LIN {X 0,Y 680.523,Z 319.435,A -85,B 0,C 180,E1 25560.421,E2 25560.421} C_VEL
LIN {X 0,Y 680.503,Z 319.465,A -85,B 0,C 180,E1 25557.305,E2 25557.305} C_VEL
LIN {X 0,Y 680.521,Z 319.439,A -85,B 0,C 180,E1 25554.266,E2 25554.266} C_VEL
LIN {X 0,Y 680.497,Z 319.465,A -85,B 0,C 180,E1 25551.21,E2 25551.21} C_VEL
LIN {X 0,Y 680.519,Z 319.439,A -85,B 0,C 180,E1 25548.215,E2 25548.215} C_VEL
LIN {X 0,Y 680.491,Z 319.465,A -85,B 0,C 180,E1 25545.1,E2 25545.1} C_VEL
LIN {X 0,Y 680.502,Z 319.438,A -85,B 0,C 180,E1 25542.198,E2 25542.198} C_VEL
LIN {X 0,Y 680.491,Z 319.464,A -85,B 0,C 180,E1 25539.08,E2 25539.08} C_VEL
LIN {X 0,Y 680.47,Z 319.444,A -85,B 0,C 180,E1 25536.35,E2 25536.35} C_VEL
LIN {X 0,Y 680.519,Z 319.455,A -85,B 0,C 180,E1 25533.281,E2 25533.281} C_VEL
LIN {X 0,Y 680.458,Z 319.465,A -85,B 0,C 180,E1 25530.51,E2 25530.51} C_VEL
LIN {X 0,Y 680.498,Z 319.446,A -85,B 0,C 180,E1 25527.766,E2 25527.766} C_VEL
LIN {X 0,Y 680.46,Z 319.462,A -85,B 0,C 180,E1 25524.726,E2 25524.726} C_VEL
LIN {X 0,Y 680.444,Z 319.466,A -85,B 0,C 180,E1 25522.21,E2 25522.21} C_VEL
LIN {X 0,Y 680.534,Z 319.527,A -85,B 0,C 180,E1 25519.314,E2 25519.314} C_VEL
LIN {X 0,Y 680.713,Z 320.476,A -85,B 0,C 180,E1 25519.153,E2 25519.153} C_VEL
LIN {X 0,Y 688.87,Z 336.842,A -85,B 0,C 180,E1 25517.211,E2 25517.211} C_VEL
LIN {X 0,Y 695.472,Z 350.637,A -85,B 0,C 180,E1 25515.703,E2 25515.703} C_VEL
LIN {X 0,Y 696.705,Z 353.093,A -85,B 0,C 180,E1 25515.558,E2 25515.558} C_VEL
LIN {X 0,Y 700.836,Z 371.518,A -85,B 0,C 180,E1 25514.953,E2 25514.953} C_VEL
LIN {X 0,Y 698.449,Z 583.894,A -85,B 0,C 180,E1 25512.191,E2 25512.191} C_VEL
LIN {X 0,Y 696.12,Z 808.395,A -85,B 0,C 180,E1 25509.364,E2 25509.364} C_VEL
LIN {X 0,Y 695.539,Z 840.013,A -85,B 0,C 180,E1 25508.911,E2 25508.911} C_VEL
LIN {X 0,Y 694.786,Z 865.208,A -85,B 0,C 180,E1 25508.397,E2 25508.397} C_VEL
LIN {X 0,Y 693.902,Z 890.782,A -85,B 0,C 180,E1 25507.726,E2 25507.726} C_VEL
LIN {X 0,Y 692.784,Z 917.463,A -85,B 0,C 180,E1 25506.847,E2 25506.847} C_VEL
LIN {X 0,Y 691.789,Z 938.354,A -85,B 0,C 180,E1 25506.033,E2 25506.033} C_VEL
LIN {X 0,Y 690.754,Z 958.67,A -85,B 0,C 180,E1 25505.129,E2 25505.129} C_VEL
LIN {X 0,Y 689.673,Z 978.671,A -85,B 0,C 180,E1 25504.122,E2 25504.122} C_VEL
LIN {X 0,Y 688.521,Z 999.46,A -85,B 0,C 180,E1 25502.946,E2 25502.946} C_VEL
LIN {X 0,Y 687.068,Z 1024.247,A -85,B 0,C 180,E1 25501.35,E2 25501.35} C_VEL
LIN {X 0,Y 685.992,Z 1043.448,A -85,B 0,C 180,E1 25499.948,E2 25499.948} C_VEL
LIN {X 0,Y 684.974,Z 1061.822,A -85,B 0,C 180,E1 25498.464,E2 25498.464} C_VEL
LIN {X 0,Y 683.767,Z 1083.482,A -85,B 0,C 180,E1 25496.498,E2 25496.498} C_VEL
LIN {X 0,Y 682.983,Z 1099.693,A -85,B 0,C 180,E1 25494.845,E2 25494.845} C_VEL
LIN {X 0,Y 682.191,Z 1116.49,A -85,B 0,C 180,E1 25492.946,E2 25492.946} C_VEL
LIN {X 0,Y 681.497,Z 1132.896,A -85,B 0,C 180,E1 25490.835,E2 25490.835} C_VEL
LIN {X 0,Y 681.036,Z 1145.574,A -85,B 0,C 180,E1 25489,E2 25489} C_VEL
LIN {X 0,Y 680.644,Z 1157.898,A -85,B 0,C 180,E1 25486.992,E2 25486.992} C_VEL
LIN {X 0,Y 680.336,Z 1169.839,A -85,B 0,C 180,E1 25484.729,E2 25484.729} C_VEL
LIN {X 0,Y 680.158,Z 1178.438,A -85,B 0,C 180,E1 25482.825,E2 25482.825} C_VEL
LIN {X 0,Y 680.019,Z 1186.223,A -85,B 0,C 180,E1 25480.82,E2 25480.82} C_VEL
LIN {X 0,Y 679.964,Z 1193.354,A -85,B 0,C 180,E1 25478.541,E2 25478.541} C_VEL
LIN {X 0,Y 679.926,Z 1198.83,A -85,B 0,C 180,E1 25476.216,E2 25476.216} C_VEL
LIN {X 0,Y 679.913,Z 1202.374,A -85,B 0,C 180,E1 25474.048,E2 25474.048} C_VEL
LIN {X 0,Y 679.907,Z 1204.494,A -85,B 0,C 180,E1 25471.77,E2 25471.77} C_VEL
LIN {X 0,Y 679.891,Z 1204.872,A -85,B 0,C 180,E1 25469.494,E2 25469.494} C_VEL
LIN {X 0,Y 679.907,Z 1203.956,A -85,B 0,C 180,E1 25467.471,E2 25467.471} C_VEL
LIN {X 0,Y 679.911,Z 1201.427,A -85,B 0,C 180,E1 25465.276,E2 25465.276} C_VEL
LIN {X 0,Y 679.933,Z 1197.151,A -85,B 0,C 180,E1 25462.989,E2 25462.989} C_VEL
LIN {X 0,Y 679.979,Z 1191.384,A -85,B 0,C 180,E1 25460.777,E2 25460.777} C_VEL
LIN {X 0,Y 680.067,Z 1184.276,A -85,B 0,C 180,E1 25458.637,E2 25458.637} C_VEL
LIN {X 0,Y 680.241,Z 1173.935,A -85,B 0,C 180,E1 25456.137,E2 25456.137} C_VEL
LIN {X 0,Y 680.464,Z 1164.535,A -85,B 0,C 180,E1 25454.226,E2 25454.226} C_VEL
LIN {X 0,Y 680.75,Z 1154.226,A -85,B 0,C 180,E1 25452.388,E2 25452.388} C_VEL
LIN {X 0,Y 681.151,Z 1141.935,A -85,B 0,C 180,E1 25450.446,E2 25450.446} C_VEL
LIN {X 0,Y 681.795,Z 1125.468,A -85,B 0,C 180,E1 25448.177,E2 25448.177} C_VEL
LIN {X 0,Y 682.44,Z 1111.066,A -85,B 0,C 180,E1 25446.423,E2 25446.423} C_VEL
LIN {X 0,Y 683.272,Z 1093.714,A -85,B 0,C 180,E1 25444.518,E2 25444.518} C_VEL
LIN {X 0,Y 684.267,Z 1074.727,A -85,B 0,C 180,E1 25442.679,E2 25442.679} C_VEL
LIN {X 0,Y 685.157,Z 1057.943,A -85,B 0,C 180,E1 25441.211,E2 25441.211} C_VEL
LIN {X 0,Y 686.262,Z 1038.582,A -85,B 0,C 180,E1 25439.679,E2 25439.679} C_VEL
LIN {X 0,Y 687.621,Z 1015.166,A -85,B 0,C 180,E1 25438.042,E2 25438.042} C_VEL
LIN {X 0,Y 688.735,Z 995.434,A -85,B 0,C 180,E1 25436.817,E2 25436.817} C_VEL
LIN {X 0,Y 689.842,Z 975.499,A -85,B 0,C 180,E1 25435.709,E2 25435.709} C_VEL
LIN {X 0,Y 691.119,Z 951.675,A -85,B 0,C 180,E1 25434.539,E2 25434.539} C_VEL
LIN {X 0,Y 692.336,Z 926.405,A -85,B 0,C 180,E1 25433.486,E2 25433.486} C_VEL
LIN {X 0,Y 693.318,Z 904.116,A -85,B 0,C 180,E1 25432.694,E2 25432.694} C_VEL
LIN {X 0,Y 694.253,Z 881.033,A -85,B 0,C 180,E1 25432.001,E2 25432.001} C_VEL
LIN {X 0,Y 695.166,Z 854.064,A -85,B 0,C 180,E1 25431.355,E2 25431.355} C_VEL
LIN {X 0,Y 695.823,Z 827.013,A -85,B 0,C 180,E1 25430.882,E2 25430.882} C_VEL
LIN {X 0,Y 698.199,Z 606.762,A -85,B 0,C 180,E1 25428.101,E2 25428.101} C_VEL
LIN {X 0,Y 700.451,Z 403.611,A -85,B 0,C 180,E1 25425.47,E2 25425.47} C_VEL
LIN {X 0,Y 700.679,Z 370.058,A -85,B 0,C 180,E1 25425.014,E2 25425.014} C_VEL
LIN {X 0,Y 696.204,Z 351.824,A -85,B 0,C 180,E1 25424.382,E2 25424.382} C_VEL
LIN {X 0,Y 694.705,Z 349.075,A -85,B 0,C 180,E1 25424.157,E2 25424.157} C_VEL
LIN {X 0,Y 686.31,Z 331.797,A -85,B 0,C 180,E1 25422.194,E2 25422.194} C_VEL
LIN {X 0,Y 681.971,Z 323.226,A -85,B 0,C 180,E1 25421.172,E2 25421.172} C_VEL
LIN {X 0,Y 680.561,Z 319.709,A -85,B 0,C 180,E1 25420.745,E2 25420.745} C_VEL
LIN {X 0,Y 680.447,Z 319.469,A -85,B 0,C 180,E1 25417.897,E2 25417.897} C_VEL
LIN {X 0,Y 680.453,Z 319.462,A -85,B 0,C 180,E1 25415.36,E2 25415.36} C_VEL
LIN {X 0,Y 680.511,Z 319.443,A -85,B 0,C 180,E1 25412.333,E2 25412.333} C_VEL
LIN {X 0,Y 680.457,Z 319.465,A -85,B 0,C 180,E1 25409.553,E2 25409.553} C_VEL
LIN {X 0,Y 680.502,Z 319.454,A -85,B 0,C 180,E1 25406.814,E2 25406.814} C_VEL
LIN {X 0,Y 680.474,Z 319.444,A -85,B 0,C 180,E1 25403.733,E2 25403.733} C_VEL
LIN {X 0,Y 680.48,Z 319.464,A -85,B 0,C 180,E1 25401.01,E2 25401.01} C_VEL
LIN {X 0,Y 680.509,Z 319.438,A -85,B 0,C 180,E1 25397.884,E2 25397.884} C_VEL
LIN {X 0,Y 680.481,Z 319.465,A -85,B 0,C 180,E1 25394.988,E2 25394.988} C_VEL
LIN {X 0,Y 680.522,Z 319.437,A -85,B 0,C 180,E1 25391.957,E2 25391.957} C_VEL
LIN {X 0,Y 680.483,Z 319.463,A -85,B 0,C 180,E1 25389.046,E2 25389.046} C_VEL
LIN {X 0,Y 680.517,Z 319.437,A -85,B 0,C 180,E1 25386.157,E2 25386.157} C_VEL
LIN {X 0,Y 680.493,Z 319.46,A -85,B 0,C 180,E1 25383.117,E2 25383.117} C_VEL
LIN {X 0,Y 680.518,Z 319.436,A -85,B 0,C 180,E1 25380.168,E2 25380.168} C_VEL
LIN {X 0,Y 680.504,Z 319.457,A -85,B 0,C 180,E1 25377.116,E2 25377.116} C_VEL
LIN {X 0,Y 680.515,Z 319.436,A -85,B 0,C 180,E1 25374.097,E2 25374.097} C_VEL
LIN {X 0,Y 680.513,Z 319.455,A -85,B 0,C 180,E1 25371.04,E2 25371.04} C_VEL
LIN {X 0,Y 680.514,Z 319.438,A -85,B 0,C 180,E1 25368.043,E2 25368.043} C_VEL
LIN {X 0,Y 680.523,Z 319.455,A -85,B 0,C 180,E1 25365.013,E2 25365.013} C_VEL
LIN {X 0,Y 680.509,Z 319.44,A -85,B 0,C 180,E1 25361.924,E2 25361.924} C_VEL
LIN {X 0,Y 680.526,Z 319.457,A -85,B 0,C 180,E1 25358.901,E2 25358.901} C_VEL
LIN {X 0,Y 680.503,Z 319.444,A -85,B 0,C 180,E1 25355.798,E2 25355.798} C_VEL
LIN {X 0,Y 680.523,Z 319.457,A -85,B 0,C 180,E1 25352.737,E2 25352.737} C_VEL
LIN {X 0,Y 680.495,Z 319.462,A -85,B 0,C 180,E1 25349.638,E2 25349.638} C_VEL
LIN {X 0,Y 680.486,Z 319.466,A -85,B 0,C 180,E1 25349.46,E2 25349.46} C_VEL
LIN {X 0,Y 679.484,Z 319.589,A -85,B 0,C 180,E1 25348.811,E2 25348.811} C_VEL
LIN {X 0,Y 673.087,Z 320.364,A -85,B 0,C 180,E1 25346.994,E2 25346.994} C_VEL
LIN {X 0,Y 672.583,Z 320.425,A -85,B 0,C 180,E1 25346.521,E2 25346.521} C_VEL
LIN {X 0,Y 672.547,Z 320.44,A -85,B 0,C 180,E1 25343.509,E2 25343.509} C_VEL
LIN {X 0,Y 672.564,Z 320.456,A -85,B 0,C 180,E1 25340.594,E2 25340.594} C_VEL
LIN {X 0,Y 672.618,Z 320.685,A -85,B 0,C 180,E1 25338.341,E2 25338.341} C_VEL
LIN {X 0,Y 674.146,Z 324.296,A -85,B 0,C 180,E1 25337.867,E2 25337.867} C_VEL
LIN {X 0,Y 680.947,Z 338.516,A -85,B 0,C 180,E1 25336.126,E2 25336.126} C_VEL
LIN {X 0,Y 687.645,Z 353.245,A -85,B 0,C 180,E1 25334.442,E2 25334.442} C_VEL
LIN {X 0,Y 688.188,Z 354.8,A -85,B 0,C 180,E1 25334.283,E2 25334.283} C_VEL
LIN {X 0,Y 686.298,Z 396.404,A -85,B 0,C 180,E1 25331.484,E2 25331.484} C_VEL
LIN {X 0,Y 690.87,Z 417.786,A -85,B 0,C 180,E1 25330.837,E2 25330.837} C_VEL
LIN {X 0,Y 688.26,Z 661.816,A -85,B 0,C 180,E1 25327.794,E2 25327.794} C_VEL
LIN {X 0,Y 686.473,Z 830.346,A -85,B 0,C 180,E1 25325.723,E2 25325.723} C_VEL
LIN {X 0,Y 685.847,Z 856.635,A -85,B 0,C 180,E1 25325.262,E2 25325.262} C_VEL
LIN {X 0,Y 685.019,Z 880.355,A -85,B 0,C 180,E1 25324.692,E2 25324.692} C_VEL
LIN {X 0,Y 684.217,Z 900.856,A -85,B 0,C 180,E1 25324.085,E2 25324.085} C_VEL
LIN {X 0,Y 683.164,Z 924.808,A -85,B 0,C 180,E1 25323.238,E2 25323.238} C_VEL
LIN {X 0,Y 681.985,Z 948.429,A -85,B 0,C 180,E1 25322.224,E2 25322.224} C_VEL
LIN {X 0,Y 680.95,Z 968.049,A -85,B 0,C 180,E1 25321.255,E2 25321.255} C_VEL
LIN {X 0,Y 679.738,Z 990.237,A -85,B 0,C 180,E1 25320.009,E2 25320.009} C_VEL
LIN {X 0,Y 678.458,Z 1011.622,A -85,B 0,C 180,E1 25318.618,E2 25318.618} C_VEL
LIN {X 0,Y 677.441,Z 1029.893,A -85,B 0,C 180,E1 25317.282,E2 25317.282} C_VEL
LIN {X 0,Y 676.241,Z 1051.038,A -85,B 0,C 180,E1 25315.532,E2 25315.532} C_VEL
LIN {X 0,Y 675.373,Z 1067.296,A -85,B 0,C 180,E1 25314.01,E2 25314.01} C_VEL
LIN {X 0,Y 674.523,Z 1084.551,A -85,B 0,C 180,E1 25312.21,E2 25312.21} C_VEL
LIN {X 0,Y 673.77,Z 1100.533,A -85,B 0,C 180,E1 25310.297,E2 25310.297} C_VEL
LIN {X 0,Y 673.204,Z 1114.293,A -85,B 0,C 180,E1 25308.443,E2 25308.443} C_VEL
LIN {X 0,Y 672.711,Z 1127.982,A -85,B 0,C 180,E1 25306.315,E2 25306.315} C_VEL
LIN {X 0,Y 672.442,Z 1137.959,A -85,B 0,C 180,E1 25304.531,E2 25304.531} C_VEL
LIN {X 0,Y 672.2,Z 1148.015,A -85,B 0,C 180,E1 25302.456,E2 25302.456} C_VEL
LIN {X 0,Y 672.044,Z 1156.61,A -85,B 0,C 180,E1 25300.285,E2 25300.285} C_VEL
LIN {X 0,Y 671.973,Z 1162.516,A -85,B 0,C 180,E1 25298.471,E2 25298.471} C_VEL
LIN {X 0,Y 671.925,Z 1167.459,A -85,B 0,C 180,E1 25296.58,E2 25296.58} C_VEL
LIN {X 0,Y 671.909,Z 1171.777,A -85,B 0,C 180,E1 25294.267,E2 25294.267} C_VEL
LIN {X 0,Y 671.913,Z 1173.902,A -85,B 0,C 180,E1 25292.388,E2 25292.388} C_VEL
LIN {X 0,Y 671.892,Z 1174.837,A -85,B 0,C 180,E1 25290.597,E2 25290.597} C_VEL
LIN {X 0,Y 671.91,Z 1174.637,A -85,B 0,C 180,E1 25288.551,E2 25288.551} C_VEL
LIN {X 0,Y 671.897,Z 1172.688,A -85,B 0,C 180,E1 25286.331,E2 25286.331} C_VEL
LIN {X 0,Y 671.909,Z 1169.91,A -85,B 0,C 180,E1 25284.535,E2 25284.535} C_VEL
LIN {X 0,Y 671.944,Z 1166.023,A -85,B 0,C 180,E1 25282.734,E2 25282.734} C_VEL
LIN {X 0,Y 672.007,Z 1159.937,A -85,B 0,C 180,E1 25280.573,E2 25280.573} C_VEL
LIN {X 0,Y 672.123,Z 1151.993,A -85,B 0,C 180,E1 25278.415,E2 25278.415} C_VEL
LIN {X 0,Y 672.271,Z 1144.372,A -85,B 0,C 180,E1 25276.672,E2 25276.672} C_VEL
LIN {X 0,Y 672.556,Z 1133.669,A -85,B 0,C 180,E1 25274.567,E2 25274.567} C_VEL
LIN {X 0,Y 672.937,Z 1121.399,A -85,B 0,C 180,E1 25272.534,E2 25272.534} C_VEL
LIN {X 0,Y 673.404,Z 1109.186,A -85,B 0,C 180,E1 25270.754,E2 25270.754} C_VEL
LIN {X 0,Y 674.119,Z 1092.876,A -85,B 0,C 180,E1 25268.668,E2 25268.668} C_VEL
LIN {X 0,Y 674.819,Z 1077.786,A -85,B 0,C 180,E1 25266.973,E2 25266.973} C_VEL
LIN {X 0,Y 675.804,Z 1059.628,A -85,B 0,C 180,E1 25265.154,E2 25265.154} C_VEL
LIN {X 0,Y 676.807,Z 1040.8,A -85,B 0,C 180,E1 25263.503,E2 25263.503} C_VEL
LIN {X 0,Y 677.936,Z 1021.383,A -85,B 0,C 180,E1 25261.982,E2 25261.982} C_VEL
LIN {X 0,Y 679.191,Z 999.206,A -85,B 0,C 180,E1 25260.466,E2 25260.466} C_VEL
LIN {X 0,Y 680.323,Z 978.831,A -85,B 0,C 180,E1 25259.239,E2 25259.239} C_VEL
LIN {X 0,Y 681.679,Z 954.593,A -85,B 0,C 180,E1 25257.975,E2 25257.975} C_VEL
LIN {X 0,Y 682.736,Z 933.698,A -85,B 0,C 180,E1 25257.039,E2 25257.039} C_VEL
LIN {X 0,Y 683.65,Z 914.34,A -85,B 0,C 180,E1 25256.287,E2 25256.287} C_VEL
LIN {X 0,Y 684.698,Z 889.896,A -85,B 0,C 180,E1 25255.48,E2 25255.48} C_VEL
LIN {X 0,Y 685.52,Z 864.903,A -85,B 0,C 180,E1 25254.831,E2 25254.831} C_VEL
LIN {X 0,Y 686.17,Z 842.781,A -85,B 0,C 180,E1 25254.384,E2 25254.384} C_VEL
LIN {X 0,Y 686.74,Z 813.095,A -85,B 0,C 180,E1 25253.957,E2 25253.957} C_VEL
LIN {X 0,Y 689.172,Z 573.619,A -85,B 0,C 180,E1 25251.027,E2 25251.027} C_VEL
LIN {X 0,Y 690.784,Z 416.524,A -85,B 0,C 180,E1 25249.05,E2 25249.05} C_VEL
LIN {X 0,Y 686.265,Z 396.184,A -85,B 0,C 180,E1 25248.417,E2 25248.417} C_VEL
LIN {X 0,Y 688.188,Z 354.854,A -85,B 0,C 180,E1 25245.631,E2 25245.631} C_VEL
LIN {X 0,Y 683.619,Z 344.296,A -85,B 0,C 180,E1 25244.459,E2 25244.459} C_VEL
LIN {X 0,Y 678.067,Z 332.508,A -85,B 0,C 180,E1 25243.059,E2 25243.059} C_VEL
LIN {X 0,Y 673.851,Z 323.857,A -85,B 0,C 180,E1 25241.979,E2 25241.979} C_VEL
LIN {X 0,Y 672.598,Z 320.636,A -85,B 0,C 180,E1 25241.546,E2 25241.546} C_VEL
LIN {X 0,Y 672.527,Z 320.454,A -85,B 0,C 180,E1 25238.751,E2 25238.751} C_VEL
LIN {X 0,Y 672.587,Z 320.447,A -85,B 0,C 180,E1 25235.855,E2 25235.855} C_VEL
LIN {X 0,Y 672.537,Z 320.433,A -85,B 0,C 180,E1 25232.86,E2 25232.86} C_VEL
LIN {X 0,Y 672.586,Z 320.436,A -85,B 0,C 180,E1 25229.968,E2 25229.968} C_VEL
LIN {X 0,Y 672.554,Z 320.449,A -85,B 0,C 180,E1 25226.87,E2 25226.87} C_VEL
LIN {X 0,Y 672.579,Z 320.427,A -85,B 0,C 180,E1 25223.897,E2 25223.897} C_VEL
LIN {X 0,Y 672.562,Z 320.449,A -85,B 0,C 180,E1 25220.754,E2 25220.754} C_VEL
LIN {X 0,Y 672.58,Z 320.428,A -85,B 0,C 180,E1 25217.744,E2 25217.744} C_VEL
LIN {X 0,Y 672.567,Z 320.447,A -85,B 0,C 180,E1 25214.64,E2 25214.64} C_VEL
LIN {X 0,Y 672.575,Z 320.431,A -85,B 0,C 180,E1 25211.567,E2 25211.567} C_VEL
LIN {X 0,Y 672.572,Z 320.445,A -85,B 0,C 180,E1 25208.464,E2 25208.464} C_VEL
LIN {X 0,Y 672.57,Z 320.431,A -85,B 0,C 180,E1 25205.46,E2 25205.46} C_VEL
LIN {X 0,Y 672.579,Z 320.445,A -85,B 0,C 180,E1 25202.386,E2 25202.386} C_VEL
LIN {X 0,Y 672.564,Z 320.432,A -85,B 0,C 180,E1 25199.319,E2 25199.319} C_VEL
LIN {X 0,Y 672.582,Z 320.447,A -85,B 0,C 180,E1 25196.249,E2 25196.249} C_VEL
LIN {X 0,Y 672.553,Z 320.433,A -85,B 0,C 180,E1 25193.169,E2 25193.169} C_VEL
LIN {X 0,Y 672.585,Z 320.446,A -85,B 0,C 180,E1 25190.156,E2 25190.156} C_VEL
LIN {X 0,Y 672.551,Z 320.434,A -85,B 0,C 180,E1 25187.114,E2 25187.114} C_VEL
LIN {X 0,Y 672.57,Z 320.448,A -85,B 0,C 180,E1 25184.213,E2 25184.213} C_VEL
LIN {X 0,Y 672.549,Z 320.438,A -85,B 0,C 180,E1 25181.089,E2 25181.089} C_VEL
LIN {X 0,Y 672.545,Z 320.448,A -85,B 0,C 180,E1 25178.272,E2 25178.272} C_VEL
LIN {X 0,Y 672.552,Z 320.451,A -85,B 0,C 180,E1 25175.077,E2 25175.077} C_VEL
LIN {X 0,Y 672.523,Z 320.437,A -85,B 0,C 180,E1 25172.362,E2 25172.362} C_VEL
LIN {X 0,Y 672.59,Z 320.454,A -85,B 0,C 180,E1 25169.4,E2 25169.4} C_VEL
LIN {X 0,Y 672.513,Z 320.445,A -85,B 0,C 180,E1 25166.52,E2 25166.52} C_VEL
LIN {X 0,Y 672.535,Z 320.433,A -85,B 0,C 180,E1 25163.826,E2 25163.826} C_VEL
LIN {X 0,Y 672.516,Z 320.44,A -85,B 0,C 180,E1 25160.7,E2 25160.7} C_VEL
LIN {X 0,Y 672.546,Z 320.693,A -85,B 0,C 180,E1 25159.954,E2 25159.954} C_VEL
LIN {X 0,Y 674.168,Z 324.332,A -85,B 0,C 180,E1 25159.487,E2 25159.487} C_VEL
LIN {X 0,Y 683.149,Z 342.282,A -85,B 0,C 180,E1 25157.338,E2 25157.338} C_VEL
LIN {X 0,Y 687.378,Z 350.803,A -85,B 0,C 180,E1 25156.395,E2 25156.395} C_VEL
LIN {X 0,Y 691.603,Z 357.548,A -85,B 0,C 180,E1 25155.925,E2 25155.925} C_VEL
LIN {X 0,Y 695.139,Z 373.566,A -85,B 0,C 180,E1 25155.394,E2 25155.394} C_VEL
LIN {X 0,Y 692.485,Z 586.297,A -85,B 0,C 180,E1 25152.607,E2 25152.607} C_VEL
LIN {X 0,Y 689.906,Z 810.507,A -85,B 0,C 180,E1 25149.761,E2 25149.761} C_VEL
LIN {X 0,Y 689.269,Z 840.637,A -85,B 0,C 180,E1 25149.32,E2 25149.32} C_VEL
LIN {X 0,Y 688.472,Z 865.187,A -85,B 0,C 180,E1 25148.815,E2 25148.815} C_VEL
LIN {X 0,Y 687.488,Z 890.734,A -85,B 0,C 180,E1 25148.142,E2 25148.142} C_VEL
LIN {X 0,Y 686.225,Z 918.038,A -85,B 0,C 180,E1 25147.235,E2 25147.235} C_VEL
LIN {X 0,Y 685.095,Z 939.48,A -85,B 0,C 180,E1 25146.39,E2 25146.39} C_VEL
LIN {X 0,Y 683.956,Z 959.717,A -85,B 0,C 180,E1 25145.477,E2 25145.477} C_VEL
LIN {X 0,Y 682.726,Z 980.329,A -85,B 0,C 180,E1 25144.424,E2 25144.424} C_VEL
LIN {X 0,Y 681.2,Z 1004.932,A -85,B 0,C 180,E1 25142.994,E2 25142.994} C_VEL
LIN {X 0,Y 679.764,Z 1026.915,A -85,B 0,C 180,E1 25141.527,E2 25141.527} C_VEL
LIN {X 0,Y 678.597,Z 1045.715,A -85,B 0,C 180,E1 25140.125,E2 25140.125} C_VEL
LIN {X 0,Y 677.318,Z 1066.77,A -85,B 0,C 180,E1 25138.376,E2 25138.376} C_VEL
LIN {X 0,Y 676.138,Z 1085.454,A -85,B 0,C 180,E1 25136.62,E2 25136.62} C_VEL
LIN {X 0,Y 675.284,Z 1101.391,A -85,B 0,C 180,E1 25134.96,E2 25134.96} C_VEL
LIN {X 0,Y 674.295,Z 1120.136,A -85,B 0,C 180,E1 25132.769,E2 25132.769} C_VEL
LIN {X 0,Y 673.636,Z 1134.462,A -85,B 0,C 180,E1 25130.869,E2 25130.869} C_VEL
LIN {X 0,Y 673.123,Z 1147.168,A -85,B 0,C 180,E1 25128.984,E2 25128.984} C_VEL
LIN {X 0,Y 672.64,Z 1160.813,A -85,B 0,C 180,E1 25126.672,E2 25126.672} C_VEL
LIN {X 0,Y 672.362,Z 1171.072,A -85,B 0,C 180,E1 25124.644,E2 25124.644} C_VEL
LIN {X 0,Y 672.176,Z 1179.154,A -85,B 0,C 180,E1 25122.805,E2 25122.805} C_VEL
LIN {X 0,Y 672.03,Z 1186.719,A -85,B 0,C 180,E1 25120.805,E2 25120.805} C_VEL
LIN {X 0,Y 671.969,Z 1193.595,A -85,B 0,C 180,E1 25118.557,E2 25118.557} C_VEL
LIN {X 0,Y 671.928,Z 1198.937,A -85,B 0,C 180,E1 25116.236,E2 25116.236} C_VEL
LIN {X 0,Y 671.915,Z 1202.371,A -85,B 0,C 180,E1 25114.096,E2 25114.096} C_VEL
LIN {X 0,Y 671.907,Z 1204.494,A -85,B 0,C 180,E1 25111.791,E2 25111.791} C_VEL
LIN {X 0,Y 671.891,Z 1204.872,A -85,B 0,C 180,E1 25109.488,E2 25109.488} C_VEL
LIN {X 0,Y 671.907,Z 1203.953,A -85,B 0,C 180,E1 25107.441,E2 25107.441} C_VEL
LIN {X 0,Y 671.914,Z 1201.427,A -85,B 0,C 180,E1 25105.22,E2 25105.22} C_VEL
LIN {X 0,Y 671.941,Z 1197.151,A -85,B 0,C 180,E1 25102.905,E2 25102.905} C_VEL
LIN {X 0,Y 671.991,Z 1191.381,A -85,B 0,C 180,E1 25100.666,E2 25100.666} C_VEL
LIN {X 0,Y 672.09,Z 1184.276,A -85,B 0,C 180,E1 25098.501,E2 25098.501} C_VEL
LIN {X 0,Y 672.277,Z 1174.339,A -85,B 0,C 180,E1 25096.058,E2 25096.058} C_VEL
LIN {X 0,Y 672.534,Z 1164.537,A -85,B 0,C 180,E1 25094.035,E2 25094.035} C_VEL
LIN {X 0,Y 672.865,Z 1154.228,A -85,B 0,C 180,E1 25092.175,E2 25092.175} C_VEL
LIN {X 0,Y 673.32,Z 1141.937,A -85,B 0,C 180,E1 25090.21,E2 25090.21} C_VEL
LIN {X 0,Y 674.025,Z 1125.804,A -85,B 0,C 180,E1 25087.956,E2 25087.956} C_VEL
LIN {X 0,Y 674.751,Z 1111.068,A -85,B 0,C 180,E1 25086.137,E2 25086.137} C_VEL
LIN {X 0,Y 675.713,Z 1093.715,A -85,B 0,C 180,E1 25084.212,E2 25084.212} C_VEL
LIN {X 0,Y 676.819,Z 1074.319,A -85,B 0,C 180,E1 25082.314,E2 25082.314} C_VEL
LIN {X 0,Y 677.817,Z 1057.656,A -85,B 0,C 180,E1 25080.845,E2 25080.845} C_VEL
LIN {X 0,Y 679.091,Z 1037.972,A -85,B 0,C 180,E1 25079.275,E2 25079.275} C_VEL
LIN {X 0,Y 680.589,Z 1014.441,A -85,B 0,C 180,E1 25077.622,E2 25077.622} C_VEL
LIN {X 0,Y 681.824,Z 994.634,A -85,B 0,C 180,E1 25076.386,E2 25076.386} C_VEL
LIN {X 0,Y 683.132,Z 973.152,A -85,B 0,C 180,E1 25075.192,E2 25075.192} C_VEL
LIN {X 0,Y 684.732,Z 946.206,A -85,B 0,C 180,E1 25073.899,E2 25073.899} C_VEL
LIN {X 0,Y 685.854,Z 925.016,A -85,B 0,C 180,E1 25073.027,E2 25073.027} C_VEL
LIN {X 0,Y 686.854,Z 904.042,A -85,B 0,C 180,E1 25072.279,E2 25072.279} C_VEL
LIN {X 0,Y 687.876,Z 880.995,A -85,B 0,C 180,E1 25071.584,E2 25071.584} C_VEL
LIN {X 0,Y 688.887,Z 854.024,A -85,B 0,C 180,E1 25070.935,E2 25070.935} C_VEL
LIN {X 0,Y 689.603,Z 827.087,A -85,B 0,C 180,E1 25070.462,E2 25070.462} C_VEL
LIN {X 0,Y 692.206,Z 609.542,A -85,B 0,C 180,E1 25067.692,E2 25067.692} C_VEL
LIN {X 0,Y 694.706,Z 406.307,A -85,B 0,C 180,E1 25065.04,E2 25065.04} C_VEL
LIN {X 0,Y 694.99,Z 372.179,A -85,B 0,C 180,E1 25064.574,E2 25064.574} C_VEL
LIN {X 0,Y 691.173,Z 356.512,A -85,B 0,C 180,E1 25064.023,E2 25064.023} C_VEL
LIN {X 0,Y 686.793,Z 349.864,A -85,B 0,C 180,E1 25063.522,E2 25063.522} C_VEL
LIN {X 0,Y 678.81,Z 333.538,A -85,B 0,C 180,E1 25061.631,E2 25061.631} C_VEL
LIN {X 0,Y 674.765,Z 325.222,A -85,B 0,C 180,E1 25060.637,E2 25060.637} C_VEL
LIN {X 0,Y 672.758,Z 321.621,A -85,B 0,C 180,E1 25060.169,E2 25060.169} C_VEL
LIN {X 0,Y 672.522,Z 320.554,A -85,B 0,C 180,E1 25059.999,E2 25059.999} C_VEL
LIN {X 0,Y 672.508,Z 320.443,A -85,B 0,C 180,E1 25057.444,E2 25057.444} C_VEL
LIN {X 0,Y 672.573,Z 320.452,A -85,B 0,C 180,E1 25054.402,E2 25054.402} C_VEL
LIN {X 0,Y 672.513,Z 320.448,A -85,B 0,C 180,E1 25051.558,E2 25051.558} C_VEL
LIN {X 0,Y 672.566,Z 320.432,A -85,B 0,C 180,E1 25048.796,E2 25048.796} C_VEL
LIN {X 0,Y 672.533,Z 320.454,A -85,B 0,C 180,E1 25045.715,E2 25045.715} C_VEL
LIN {X 0,Y 672.545,Z 320.429,A -85,B 0,C 180,E1 25042.925,E2 25042.925} C_VEL
LIN {X 0,Y 672.55,Z 320.447,A -85,B 0,C 180,E1 25039.724,E2 25039.724} C_VEL
LIN {X 0,Y 672.549,Z 320.434,A -85,B 0,C 180,E1 25036.853,E2 25036.853} C_VEL
LIN {X 0,Y 672.564,Z 320.44,A -85,B 0,C 180,E1 25033.673,E2 25033.673} C_VEL
LIN {X 0,Y 672.562,Z 320.438,A -85,B 0,C 180,E1 25030.676,E2 25030.676} C_VEL
LIN {X 0,Y 672.567,Z 320.437,A -85,B 0,C 180,E1 25027.517,E2 25027.517} C_VEL
LIN {X 0,Y 672.577,Z 320.439,A -85,B 0,C 180,E1 25024.434,E2 25024.434} C_VEL
LIN {X 0,Y 672.565,Z 320.44,A -85,B 0,C 180,E1 25021.278,E2 25021.278} C_VEL
LIN {X 0,Y 672.581,Z 320.438,A -85,B 0,C 180,E1 25018.211,E2 25018.211} C_VEL
LIN {X 0,Y 672.57,Z 320.441,A -85,B 0,C 180,E1 25015.139,E2 25015.139} C_VEL
LIN {X 0,Y 672.576,Z 320.437,A -85,B 0,C 180,E1 25012.053,E2 25012.053} C_VEL
LIN {X 0,Y 672.577,Z 320.44,A -85,B 0,C 180,E1 25009.03,E2 25009.03} C_VEL
LIN {X 0,Y 672.574,Z 320.439,A -85,B 0,C 180,E1 25005.976,E2 25005.976} C_VEL
LIN {X 0,Y 672.581,Z 320.441,A -85,B 0,C 180,E1 25002.881,E2 25002.881} C_VEL
LIN {X 0,Y 672.566,Z 320.448,A -85,B 0,C 180,E1 24999.824,E2 24999.824} C_VEL
LIN {X 0,Y 672.584,Z 320.433,A -85,B 0,C 180,E1 24996.799,E2 24996.799} C_VEL
LIN {X 0,Y 672.561,Z 320.455,A -85,B 0,C 180,E1 24993.697,E2 24993.697} C_VEL
LIN {X 0,Y 672.583,Z 320.423,A -85,B 0,C 180,E1 24990.718,E2 24990.718} C_VEL
LIN {X 0,Y 672.554,Z 320.438,A -85,B 0,C 180,E1 24987.612,E2 24987.612} C_VEL
LIN {X 0,Y 672.583,Z 320.425,A -85,B 0,C 180,E1 24986.521,E2 24986.521} C_VEL
LIN {X 0,Y 671.626,Z 320.553,A -85,B 0,C 180,E1 24985.865,E2 24985.865} C_VEL
LIN {X 0,Y 665.171,Z 321.371,A -85,B 0,C 180,E1 24984.026,E2 24984.026} C_VEL
LIN {X 0,Y 664.611,Z 321.428,A -85,B 0,C 180,E1 24983.548,E2 24983.548} C_VEL
LIN {X 0,Y 664.622,Z 321.446,A -85,B 0,C 180,E1 24980.649,E2 24980.649} C_VEL
LIN {X 0,Y 664.625,Z 321.671,A -85,B 0,C 180,E1 24979.063,E2 24979.063} C_VEL
LIN {X 0,Y 665.851,Z 324.803,A -85,B 0,C 180,E1 24978.644,E2 24978.644} C_VEL
LIN {X 0,Y 667.233,Z 327.461,A -85,B 0,C 180,E1 24978.29,E2 24978.29} C_VEL
LIN {X 0,Y 674.93,Z 343.383,A -85,B 0,C 180,E1 24976.299,E2 24976.299} C_VEL
LIN {X 0,Y 681.749,Z 358.539,A -85,B 0,C 180,E1 24974.552,E2 24974.552} C_VEL
LIN {X 0,Y 679.872,Z 396.006,A -85,B 0,C 180,E1 24972.003,E2 24972.003} C_VEL
LIN {X 0,Y 684.795,Z 419.668,A -85,B 0,C 180,E1 24971.253,E2 24971.253} C_VEL
LIN {X 0,Y 681.927,Z 662.857,A -85,B 0,C 180,E1 24968.195,E2 24968.195} C_VEL
LIN {X 0,Y 679.973,Z 830.389,A -85,B 0,C 180,E1 24966.118,E2 24966.118} C_VEL
LIN {X 0,Y 679.284,Z 856.789,A -85,B 0,C 180,E1 24965.651,E2 24965.651} C_VEL
LIN {X 0,Y 678.399,Z 880.265,A -85,B 0,C 180,E1 24965.083,E2 24965.083} C_VEL
LIN {X 0,Y 677.555,Z 900.132,A -85,B 0,C 180,E1 24964.493,E2 24964.493} C_VEL
LIN {X 0,Y 676.554,Z 921.013,A -85,B 0,C 180,E1 24963.758,E2 24963.758} C_VEL
LIN {X 0,Y 675.146,Z 946.823,A -85,B 0,C 180,E1 24962.671,E2 24962.671} C_VEL
LIN {X 0,Y 673.985,Z 966.896,A -85,B 0,C 180,E1 24961.68,E2 24961.68} C_VEL
LIN {X 0,Y 672.691,Z 988.65,A -85,B 0,C 180,E1 24960.455,E2 24960.455} C_VEL
LIN {X 0,Y 671.259,Z 1010.619,A -85,B 0,C 180,E1 24959.028,E2 24959.028} C_VEL
LIN {X 0,Y 670.119,Z 1028.755,A -85,B 0,C 180,E1 24957.697,E2 24957.697} C_VEL
LIN {X 0,Y 668.851,Z 1049.524,A -85,B 0,C 180,E1 24955.977,E2 24955.977} C_VEL
LIN {X 0,Y 667.801,Z 1066.689,A -85,B 0,C 180,E1 24954.362,E2 24954.362} C_VEL
LIN {X 0,Y 666.881,Z 1083.731,A -85,B 0,C 180,E1 24952.571,E2 24952.571} C_VEL
LIN {X 0,Y 666.024,Z 1099.653,A -85,B 0,C 180,E1 24950.659,E2 24950.659} C_VEL
LIN {X 0,Y 665.439,Z 1112.388,A -85,B 0,C 180,E1 24948.939,E2 24948.939} C_VEL
LIN {X 0,Y 664.887,Z 1126.424,A -85,B 0,C 180,E1 24946.782,E2 24946.782} C_VEL
LIN {X 0,Y 664.524,Z 1137.377,A -85,B 0,C 180,E1 24944.821,E2 24944.821} C_VEL
LIN {X 0,Y 664.27,Z 1146.802,A -85,B 0,C 180,E1 24942.872,E2 24942.872} C_VEL
LIN {X 0,Y 664.072,Z 1156.003,A -85,B 0,C 180,E1 24940.585,E2 24940.585} C_VEL
LIN {X 0,Y 663.985,Z 1162.007,A -85,B 0,C 180,E1 24938.748,E2 24938.748} C_VEL
LIN {X 0,Y 663.93,Z 1166.634,A -85,B 0,C 180,E1 24937.007,E2 24937.007} C_VEL
LIN {X 0,Y 663.918,Z 1170.382,A -85,B 0,C 180,E1 24935.185,E2 24935.185} C_VEL
LIN {X 0,Y 663.902,Z 1173.563,A -85,B 0,C 180,E1 24932.849,E2 24932.849} C_VEL
LIN {X 0,Y 663.904,Z 1174.77,A -85,B 0,C 180,E1 24930.863,E2 24930.863} C_VEL
LIN {X 0,Y 663.908,Z 1174.771,A -85,B 0,C 180,E1 24929.051,E2 24929.051} C_VEL
LIN {X 0,Y 663.908,Z 1173.5,A -85,B 0,C 180,E1 24926.979,E2 24926.979} C_VEL
LIN {X 0,Y 663.921,Z 1170.387,A -85,B 0,C 180,E1 24924.729,E2 24924.729} C_VEL
LIN {X 0,Y 663.935,Z 1166.642,A -85,B 0,C 180,E1 24922.907,E2 24922.907} C_VEL
LIN {X 0,Y 663.98,Z 1162.017,A -85,B 0,C 180,E1 24921.165,E2 24921.165} C_VEL
LIN {X 0,Y 664.074,Z 1155.402,A -85,B 0,C 180,E1 24919.152,E2 24919.152} C_VEL
LIN {X 0,Y 664.284,Z 1146.059,A -85,B 0,C 180,E1 24916.876,E2 24916.876} C_VEL
LIN {X 0,Y 664.53,Z 1136.918,A -85,B 0,C 180,E1 24915.001,E2 24915.001} C_VEL
LIN {X 0,Y 664.936,Z 1125.384,A -85,B 0,C 180,E1 24912.949,E2 24912.949} C_VEL
LIN {X 0,Y 665.471,Z 1111.749,A -85,B 0,C 180,E1 24910.88,E2 24910.88} C_VEL
LIN {X 0,Y 666.09,Z 1098.222,A -85,B 0,C 180,E1 24909.068,E2 24909.068} C_VEL
LIN {X 0,Y 667.03,Z 1080.47,A -85,B 0,C 180,E1 24906.985,E2 24906.985} C_VEL
LIN {X 0,Y 667.887,Z 1065.256,A -85,B 0,C 180,E1 24905.406,E2 24905.406} C_VEL
LIN {X 0,Y 669.056,Z 1046.328,A -85,B 0,C 180,E1 24903.65,E2 24903.65} C_VEL
LIN {X 0,Y 670.233,Z 1026.859,A -85,B 0,C 180,E1 24902.067,E2 24902.067} C_VEL
LIN {X 0,Y 671.598,Z 1006.144,A -85,B 0,C 180,E1 24900.571,E2 24900.571} C_VEL
LIN {X 0,Y 672.963,Z 983.695,A -85,B 0,C 180,E1 24899.163,E2 24899.163} C_VEL
LIN {X 0,Y 674.202,Z 963.078,A -85,B 0,C 180,E1 24898.03,E2 24898.03} C_VEL
LIN {X 0,Y 675.653,Z 938.298,A -85,B 0,C 180,E1 24896.857,E2 24896.857} C_VEL
LIN {X 0,Y 676.699,Z 918.18,A -85,B 0,C 180,E1 24896.046,E2 24896.046} C_VEL
LIN {X 0,Y 677.646,Z 898.305,A -85,B 0,C 180,E1 24895.359,E2 24895.359} C_VEL
LIN {X 0,Y 678.55,Z 876.929,A -85,B 0,C 180,E1 24894.736,E2 24894.736} C_VEL
LIN {X 0,Y 679.442,Z 850.641,A -85,B 0,C 180,E1 24894.135,E2 24894.135} C_VEL
LIN {X 0,Y 680.004,Z 827.551,A -85,B 0,C 180,E1 24893.75,E2 24893.75} C_VEL
LIN {X 0,Y 682.758,Z 590.882,A -85,B 0,C 180,E1 24890.82,E2 24890.82} C_VEL
LIN {X 0,Y 684.719,Z 418.431,A -85,B 0,C 180,E1 24888.634,E2 24888.634} C_VEL
LIN {X 0,Y 679.864,Z 395.593,A -85,B 0,C 180,E1 24887.884,E2 24887.884} C_VEL
LIN {X 0,Y 681.751,Z 358.545,A -85,B 0,C 180,E1 24885.359,E2 24885.359} C_VEL
LIN {X 0,Y 674.004,Z 341.395,A -85,B 0,C 180,E1 24883.372,E2 24883.372} C_VEL
LIN {X 0,Y 666.478,Z 325.683,A -85,B 0,C 180,E1 24881.4,E2 24881.4} C_VEL
LIN {X 0,Y 664.739,Z 322.284,A -85,B 0,C 180,E1 24880.934,E2 24880.934} C_VEL
LIN {X 0,Y 664.597,Z 321.525,A -85,B 0,C 180,E1 24880.765,E2 24880.765} C_VEL
LIN {X 0,Y 664.648,Z 321.413,A -85,B 0,C 180,E1 24877.834,E2 24877.834} C_VEL
LIN {X 0,Y 664.596,Z 321.445,A -85,B 0,C 180,E1 24874.87,E2 24874.87} C_VEL
LIN {X 0,Y 664.645,Z 321.429,A -85,B 0,C 180,E1 24871.955,E2 24871.955} C_VEL
LIN {X 0,Y 664.607,Z 321.413,A -85,B 0,C 180,E1 24868.878,E2 24868.878} C_VEL
LIN {X 0,Y 664.644,Z 321.439,A -85,B 0,C 180,E1 24865.893,E2 24865.893} C_VEL
LIN {X 0,Y 664.615,Z 321.427,A -85,B 0,C 180,E1 24862.746,E2 24862.746} C_VEL
LIN {X 0,Y 664.644,Z 321.424,A -85,B 0,C 180,E1 24859.785,E2 24859.785} C_VEL
LIN {X 0,Y 664.629,Z 321.431,A -85,B 0,C 180,E1 24856.699,E2 24856.699} C_VEL
LIN {X 0,Y 664.639,Z 321.417,A -85,B 0,C 180,E1 24853.631,E2 24853.631} C_VEL
LIN {X 0,Y 664.629,Z 321.431,A -85,B 0,C 180,E1 24850.488,E2 24850.488} C_VEL
LIN {X 0,Y 664.63,Z 321.414,A -85,B 0,C 180,E1 24847.434,E2 24847.434} C_VEL
LIN {X 0,Y 664.637,Z 321.429,A -85,B 0,C 180,E1 24844.4,E2 24844.4} C_VEL
LIN {X 0,Y 664.627,Z 321.419,A -85,B 0,C 180,E1 24841.379,E2 24841.379} C_VEL
LIN {X 0,Y 664.642,Z 321.428,A -85,B 0,C 180,E1 24838.276,E2 24838.276} C_VEL
LIN {X 0,Y 664.621,Z 321.423,A -85,B 0,C 180,E1 24835.254,E2 24835.254} C_VEL
LIN {X 0,Y 664.648,Z 321.424,A -85,B 0,C 180,E1 24832.218,E2 24832.218} C_VEL
LIN {X 0,Y 664.615,Z 321.424,A -85,B 0,C 180,E1 24829.16,E2 24829.16} C_VEL
LIN {X 0,Y 664.643,Z 321.427,A -85,B 0,C 180,E1 24826.161,E2 24826.161} C_VEL
LIN {X 0,Y 664.604,Z 321.421,A -85,B 0,C 180,E1 24823.03,E2 24823.03} C_VEL
LIN {X 0,Y 664.631,Z 321.434,A -85,B 0,C 180,E1 24820.094,E2 24820.094} C_VEL
LIN {X 0,Y 664.6,Z 321.416,A -85,B 0,C 180,E1 24816.973,E2 24816.973} C_VEL
LIN {X 0,Y 664.605,Z 321.442,A -85,B 0,C 180,E1 24814.132,E2 24814.132} C_VEL
LIN {X 0,Y 664.599,Z 321.427,A -85,B 0,C 180,E1 24810.925,E2 24810.925} C_VEL
LIN {X 0,Y 664.577,Z 321.433,A -85,B 0,C 180,E1 24808.326,E2 24808.326} C_VEL
LIN {X 0,Y 664.647,Z 321.444,A -85,B 0,C 180,E1 24805.343,E2 24805.343} C_VEL
LIN {X 0,Y 664.567,Z 321.431,A -85,B 0,C 180,E1 24802.457,E2 24802.457} C_VEL
LIN {X 0,Y 664.614,Z 321.699,A -85,B 0,C 180,E1 24800.673,E2 24800.673} C_VEL
LIN {X 0,Y 665.982,Z 325.074,A -85,B 0,C 180,E1 24800.236,E2 24800.236} C_VEL
LIN {X 0,Y 667.367,Z 327.783,A -85,B 0,C 180,E1 24799.89,E2 24799.89} C_VEL
LIN {X 0,Y 669.501,Z 331.879,A -85,B 0,C 180,E1 24799.371,E2 24799.371} C_VEL
LIN {X 0,Y 677.617,Z 348.164,A -85,B 0,C 180,E1 24797.418,E2 24797.418} C_VEL
LIN {X 0,Y 679.343,Z 351.296,A -85,B 0,C 180,E1 24797.099,E2 24797.099} C_VEL
LIN {X 0,Y 686.562,Z 362.132,A -85,B 0,C 180,E1 24796.294,E2 24796.294} C_VEL
LIN {X 0,Y 689.482,Z 375.729,A -85,B 0,C 180,E1 24795.841,E2 24795.841} C_VEL
LIN {X 0,Y 686.566,Z 588.197,A -85,B 0,C 180,E1 24793.036,E2 24793.036} C_VEL
LIN {X 0,Y 683.727,Z 812.543,A -85,B 0,C 180,E1 24790.166,E2 24790.166} C_VEL
LIN {X 0,Y 683.03,Z 841.424,A -85,B 0,C 180,E1 24789.733,E2 24789.733} C_VEL
LIN {X 0,Y 682.179,Z 865.558,A -85,B 0,C 180,E1 24789.231,E2 24789.231} C_VEL
LIN {X 0,Y 681.092,Z 891.252,A -85,B 0,C 180,E1 24788.549,E2 24788.549} C_VEL
LIN {X 0,Y 679.738,Z 917.902,A -85,B 0,C 180,E1 24787.657,E2 24787.657} C_VEL
LIN {X 0,Y 678.491,Z 939.477,A -85,B 0,C 180,E1 24786.802,E2 24786.802} C_VEL
LIN {X 0,Y 677.244,Z 959.713,A -85,B 0,C 180,E1 24785.882,E2 24785.882} C_VEL
LIN {X 0,Y 675.886,Z 980.554,A -85,B 0,C 180,E1 24784.809,E2 24784.809} C_VEL
LIN {X 0,Y 674.236,Z 1004.93,A -85,B 0,C 180,E1 24783.379,E2 24783.379} C_VEL
LIN {X 0,Y 672.656,Z 1026.64,A -85,B 0,C 180,E1 24781.92,E2 24781.92} C_VEL
LIN {X 0,Y 671.371,Z 1045.265,A -85,B 0,C 180,E1 24780.521,E2 24780.521} C_VEL
LIN {X 0,Y 669.98,Z 1066.199,A -85,B 0,C 180,E1 24778.77,E2 24778.77} C_VEL
LIN {X 0,Y 668.656,Z 1085.187,A -85,B 0,C 180,E1 24776.97,E2 24776.97} C_VEL
LIN {X 0,Y 667.707,Z 1100.543,A -85,B 0,C 180,E1 24775.358,E2 24775.358} C_VEL
LIN {X 0,Y 666.72,Z 1118.006,A -85,B 0,C 180,E1 24773.323,E2 24773.323} C_VEL
LIN {X 0,Y 665.877,Z 1133.819,A -85,B 0,C 180,E1 24771.216,E2 24771.216} C_VEL
LIN {X 0,Y 665.316,Z 1146.015,A -85,B 0,C 180,E1 24769.398,E2 24769.398} C_VEL
LIN {X 0,Y 664.821,Z 1158.889,A -85,B 0,C 180,E1 24767.234,E2 24767.234} C_VEL
LIN {X 0,Y 664.424,Z 1170.663,A -85,B 0,C 180,E1 24764.912,E2 24764.912} C_VEL
LIN {X 0,Y 664.224,Z 1178.797,A -85,B 0,C 180,E1 24763.05,E2 24763.05} C_VEL
LIN {X 0,Y 664.054,Z 1186.419,A -85,B 0,C 180,E1 24761.024,E2 24761.024} C_VEL
LIN {X 0,Y 663.977,Z 1193.595,A -85,B 0,C 180,E1 24758.661,E2 24758.661} C_VEL
LIN {X 0,Y 663.932,Z 1198.968,A -85,B 0,C 180,E1 24756.293,E2 24756.293} C_VEL
LIN {X 0,Y 663.915,Z 1202.482,A -85,B 0,C 180,E1 24754.059,E2 24754.059} C_VEL
LIN {X 0,Y 663.907,Z 1204.549,A -85,B 0,C 180,E1 24751.726,E2 24751.726} C_VEL
LIN {X 0,Y 663.891,Z 1204.872,A -85,B 0,C 180,E1 24749.482,E2 24749.482} C_VEL
LIN {X 0,Y 663.908,Z 1203.95,A -85,B 0,C 180,E1 24747.41,E2 24747.41} C_VEL
LIN {X 0,Y 663.917,Z 1201.427,A -85,B 0,C 180,E1 24745.162,E2 24745.162} C_VEL
LIN {X 0,Y 663.947,Z 1197.151,A -85,B 0,C 180,E1 24742.819,E2 24742.819} C_VEL
LIN {X 0,Y 664.001,Z 1191.281,A -85,B 0,C 180,E1 24740.519,E2 24740.519} C_VEL
LIN {X 0,Y 664.109,Z 1183.958,A -85,B 0,C 180,E1 24738.272,E2 24738.272} C_VEL
LIN {X 0,Y 664.345,Z 1173.758,A -85,B 0,C 180,E1 24735.76,E2 24735.76} C_VEL
LIN {X 0,Y 664.618,Z 1164.073,A -85,B 0,C 180,E1 24733.75,E2 24733.75} C_VEL
LIN {X 0,Y 665.008,Z 1153.637,A -85,B 0,C 180,E1 24731.854,E2 24731.854} C_VEL
LIN {X 0,Y 665.631,Z 1139.563,A -85,B 0,C 180,E1 24729.604,E2 24729.604} C_VEL
LIN {X 0,Y 666.363,Z 1124.398,A -85,B 0,C 180,E1 24727.503,E2 24727.503} C_VEL
LIN {X 0,Y 667.166,Z 1109.51,A -85,B 0,C 180,E1 24725.66,E2 24725.66} C_VEL
LIN {X 0,Y 668.347,Z 1090.656,A -85,B 0,C 180,E1 24723.583,E2 24723.583} C_VEL
LIN {X 0,Y 669.436,Z 1073.304,A -85,B 0,C 180,E1 24721.885,E2 24721.885} C_VEL
LIN {X 0,Y 670.617,Z 1056.207,A -85,B 0,C 180,E1 24720.373,E2 24720.373} C_VEL
LIN {X 0,Y 672.189,Z 1034.195,A -85,B 0,C 180,E1 24718.626,E2 24718.626} C_VEL
LIN {X 0,Y 673.616,Z 1013.164,A -85,B 0,C 180,E1 24717.156,E2 24717.156} C_VEL
LIN {X 0,Y 674.997,Z 993.059,A -85,B 0,C 180,E1 24715.901,E2 24715.901} C_VEL
LIN {X 0,Y 676.709,Z 968.642,A -85,B 0,C 180,E1 24714.553,E2 24714.553} C_VEL
LIN {X 0,Y 678.239,Z 943.974,A -85,B 0,C 180,E1 24713.393,E2 24713.393} C_VEL
LIN {X 0,Y 679.404,Z 923.868,A -85,B 0,C 180,E1 24712.568,E2 24712.568} C_VEL
LIN {X 0,Y 680.472,Z 903.027,A -85,B 0,C 180,E1 24711.826,E2 24711.826} C_VEL
LIN {X 0,Y 681.605,Z 879.602,A -85,B 0,C 180,E1 24711.122,E2 24711.122} C_VEL
LIN {X 0,Y 682.719,Z 851.746,A -85,B 0,C 180,E1 24710.463,E2 24710.463} C_VEL
LIN {X 0,Y 683.44,Z 826.197,A -85,B 0,C 180,E1 24710.021,E2 24710.021} C_VEL
LIN {X 0,Y 686.286,Z 609.434,A -85,B 0,C 180,E1 24707.239,E2 24707.239} C_VEL
LIN {X 0,Y 689.038,Z 406.266,A -85,B 0,C 180,E1 24704.567,E2 24704.567} C_VEL
LIN {X 0,Y 689.343,Z 374.303,A -85,B 0,C 180,E1 24704.126,E2 24704.126} C_VEL
LIN {X 0,Y 686.167,Z 361.224,A -85,B 0,C 180,E1 24703.658,E2 24703.658} C_VEL
LIN {X 0,Y 678.452,Z 349.943,A -85,B 0,C 180,E1 24702.783,E2 24702.783} C_VEL
LIN {X 0,Y 672.688,Z 338.298,A -85,B 0,C 180,E1 24701.411,E2 24701.411} C_VEL
LIN {X 0,Y 668.468,Z 329.737,A -85,B 0,C 180,E1 24700.367,E2 24700.367} C_VEL
LIN {X 0,Y 665.973,Z 325.066,A -85,B 0,C 180,E1 24699.762,E2 24699.762} C_VEL
LIN {X 0,Y 664.602,Z 321.608,A -85,B 0,C 180,E1 24699.301,E2 24699.301} C_VEL
LIN {X 0,Y 664.604,Z 321.418,A -85,B 0,C 180,E1 24696.247,E2 24696.247} C_VEL
LIN {X 0,Y 664.571,Z 321.432,A -85,B 0,C 180,E1 24693.517,E2 24693.517} C_VEL
LIN {X 0,Y 664.653,Z 321.443,A -85,B 0,C 180,E1 24690.563,E2 24690.563} C_VEL
LIN {X 0,Y 664.581,Z 321.424,A -85,B 0,C 180,E1 24687.605,E2 24687.605} C_VEL
LIN {X 0,Y 664.621,Z 321.434,A -85,B 0,C 180,E1 24684.818,E2 24684.818} C_VEL
LIN {X 0,Y 664.604,Z 321.437,A -85,B 0,C 180,E1 24681.722,E2 24681.722} C_VEL
LIN {X 0,Y 664.612,Z 321.424,A -85,B 0,C 180,E1 24678.861,E2 24678.861} C_VEL
LIN {X 0,Y 664.615,Z 321.439,A -85,B 0,C 180,E1 24675.623,E2 24675.623} C_VEL
LIN {X 0,Y 664.622,Z 321.416,A -85,B 0,C 180,E1 24672.689,E2 24672.689} C_VEL
LIN {X 0,Y 664.623,Z 321.437,A -85,B 0,C 180,E1 24669.526,E2 24669.526} C_VEL
LIN {X 0,Y 664.638,Z 321.411,A -85,B 0,C 180,E1 24666.479,E2 24666.479} C_VEL
LIN {X 0,Y 664.628,Z 321.436,A -85,B 0,C 180,E1 24663.364,E2 24663.364} C_VEL
LIN {X 0,Y 664.644,Z 321.409,A -85,B 0,C 180,E1 24660.259,E2 24660.259} C_VEL
LIN {X 0,Y 664.627,Z 321.435,A -85,B 0,C 180,E1 24657.122,E2 24657.122} C_VEL
LIN {X 0,Y 664.638,Z 321.409,A -85,B 0,C 180,E1 24654.128,E2 24654.128} C_VEL
LIN {X 0,Y 664.633,Z 321.433,A -85,B 0,C 180,E1 24650.998,E2 24650.998} C_VEL
LIN {X 0,Y 664.629,Z 321.409,A -85,B 0,C 180,E1 24647.924,E2 24647.924} C_VEL
LIN {X 0,Y 664.641,Z 321.434,A -85,B 0,C 180,E1 24644.914,E2 24644.914} C_VEL
LIN {X 0,Y 664.627,Z 321.412,A -85,B 0,C 180,E1 24641.855,E2 24641.855} C_VEL
LIN {X 0,Y 664.647,Z 321.436,A -85,B 0,C 180,E1 24638.835,E2 24638.835} C_VEL
LIN {X 0,Y 664.621,Z 321.417,A -85,B 0,C 180,E1 24635.74,E2 24635.74} C_VEL
LIN {X 0,Y 664.646,Z 321.436,A -85,B 0,C 180,E1 24632.688,E2 24632.688} C_VEL
LIN {X 0,Y 664.617,Z 321.436,A -85,B 0,C 180,E1 24629.635,E2 24629.635} C_VEL
LIN {X 0,Y 664.639,Z 321.412,A -85,B 0,C 180,E1 24626.61,E2 24626.61} C_VEL
LIN {X 0,Y 664.611,Z 321.428,A -85,B 0,C 180,E1 24623.548,E2 24623.548} C_VEL
LIN {X 0,Y 663.588,Z 321.556,A -85,B 0,C 180,E1 24622.884,E2 24622.884} C_VEL
LIN {X 0,Y 657.182,Z 322.381,A -85,B 0,C 180,E1 24621.022,E2 24621.022} C_VEL
LIN {X 0,Y 656.692,Z 322.429,A -85,B 0,C 180,E1 24620.538,E2 24620.538} C_VEL
LIN {X 0,Y 656.738,Z 322.699,A -85,B 0,C 180,E1 24619.793,E2 24619.793} C_VEL
LIN {X 0,Y 658.13,Z 326.13,A -85,B 0,C 180,E1 24619.324,E2 24619.324} C_VEL
LIN {X 0,Y 663.199,Z 336.23,A -85,B 0,C 180,E1 24617.978,E2 24617.978} C_VEL
LIN {X 0,Y 670.747,Z 352.221,A -85,B 0,C 180,E1 24615.999,E2 24615.999} C_VEL
LIN {X 0,Y 675.345,Z 362.887,A -85,B 0,C 180,E1 24614.779,E2 24614.779} C_VEL
LIN {X 0,Y 673.591,Z 396.11,A -85,B 0,C 180,E1 24612.514,E2 24612.514} C_VEL
LIN {X 0,Y 678.98,Z 421.446,A -85,B 0,C 180,E1 24611.698,E2 24611.698} C_VEL
LIN {X 0,Y 676.09,Z 626.773,A -85,B 0,C 180,E1 24609.068,E2 24609.068} C_VEL
LIN {X 0,Y 673.505,Z 830.325,A -85,B 0,C 180,E1 24606.522,E2 24606.522} C_VEL
LIN {X 0,Y 672.753,Z 856.894,A -85,B 0,C 180,E1 24606.049,E2 24606.049} C_VEL
LIN {X 0,Y 671.819,Z 879.981,A -85,B 0,C 180,E1 24605.488,E2 24605.488} C_VEL
LIN {X 0,Y 670.928,Z 899.409,A -85,B 0,C 180,E1 24604.909,E2 24604.909} C_VEL
LIN {X 0,Y 669.912,Z 919.031,A -85,B 0,C 180,E1 24604.22,E2 24604.22} C_VEL
LIN {X 0,Y 668.562,Z 942.714,A -85,B 0,C 180,E1 24603.244,E2 24603.244} C_VEL
LIN {X 0,Y 667.045,Z 966.003,A -85,B 0,C 180,E1 24602.099,E2 24602.099} C_VEL
LIN {X 0,Y 665.719,Z 986.42,A -85,B 0,C 180,E1 24600.949,E2 24600.949} C_VEL
LIN {X 0,Y 664.116,Z 1009.629,A -85,B 0,C 180,E1 24599.444,E2 24599.444} C_VEL
LIN {X 0,Y 662.81,Z 1028.155,A -85,B 0,C 180,E1 24598.078,E2 24598.078} C_VEL
LIN {X 0,Y 661.494,Z 1048.009,A -85,B 0,C 180,E1 24596.433,E2 24596.433} C_VEL
LIN {X 0,Y 660.243,Z 1066.503,A -85,B 0,C 180,E1 24594.679,E2 24594.679} C_VEL
LIN {X 0,Y 659.246,Z 1082.889,A -85,B 0,C 180,E1 24592.942,E2 24592.942} C_VEL
LIN {X 0,Y 658.258,Z 1099.659,A -85,B 0,C 180,E1 24590.914,E2 24590.914} C_VEL
LIN {X 0,Y 657.62,Z 1112.391,A -85,B 0,C 180,E1 24589.173,E2 24589.173} C_VEL
LIN {X 0,Y 657.006,Z 1126.429,A -85,B 0,C 180,E1 24586.99,E2 24586.99} C_VEL
LIN {X 0,Y 656.59,Z 1137.382,A -85,B 0,C 180,E1 24585.004,E2 24585.004} C_VEL
LIN {X 0,Y 656.316,Z 1146.398,A -85,B 0,C 180,E1 24583.12,E2 24583.12} C_VEL
LIN {X 0,Y 656.089,Z 1155.701,A -85,B 0,C 180,E1 24580.804,E2 24580.804} C_VEL
LIN {X 0,Y 655.996,Z 1162.009,A -85,B 0,C 180,E1 24578.856,E2 24578.856} C_VEL
LIN {X 0,Y 655.939,Z 1166.656,A -85,B 0,C 180,E1 24577.084,E2 24577.084} C_VEL
LIN {X 0,Y 655.919,Z 1170.542,A -85,B 0,C 180,E1 24575.16,E2 24575.16} C_VEL
LIN {X 0,Y 655.902,Z 1173.631,A -85,B 0,C 180,E1 24572.796,E2 24572.796} C_VEL
LIN {X 0,Y 655.904,Z 1174.77,A -85,B 0,C 180,E1 24570.874,E2 24570.874} C_VEL
LIN {X 0,Y 655.909,Z 1174.771,A -85,B 0,C 180,E1 24569.039,E2 24569.039} C_VEL
LIN {X 0,Y 655.908,Z 1173.5,A -85,B 0,C 180,E1 24566.942,E2 24566.942} C_VEL
LIN {X 0,Y 655.918,Z 1170.386,A -85,B 0,C 180,E1 24564.665,E2 24564.665} C_VEL
LIN {X 0,Y 655.945,Z 1166.641,A -85,B 0,C 180,E1 24562.82,E2 24562.82} C_VEL
LIN {X 0,Y 656,Z 1161.76,A -85,B 0,C 180,E1 24560.968,E2 24560.968} C_VEL
LIN {X 0,Y 656.118,Z 1154.463,A -85,B 0,C 180,E1 24558.752,E2 24558.752} C_VEL
LIN {X 0,Y 656.333,Z 1145.592,A -85,B 0,C 180,E1 24556.611,E2 24556.611} C_VEL
LIN {X 0,Y 656.612,Z 1136.452,A -85,B 0,C 180,E1 24554.726,E2 24554.726} C_VEL
LIN {X 0,Y 657.089,Z 1124.258,A -85,B 0,C 180,E1 24552.556,E2 24552.556} C_VEL
LIN {X 0,Y 657.68,Z 1111.107,A -85,B 0,C 180,E1 24550.552,E2 24550.552} C_VEL
LIN {X 0,Y 658.435,Z 1096.802,A -85,B 0,C 180,E1 24548.626,E2 24548.626} C_VEL
LIN {X 0,Y 659.368,Z 1080.315,A -85,B 0,C 180,E1 24546.685,E2 24546.685} C_VEL
LIN {X 0,Y 660.338,Z 1065.156,A -85,B 0,C 180,E1 24545.096,E2 24545.096} C_VEL
LIN {X 0,Y 661.606,Z 1046.321,A -85,B 0,C 180,E1 24543.33,E2 24543.33} C_VEL
LIN {X 0,Y 662.884,Z 1027.12,A -85,B 0,C 180,E1 24541.752,E2 24541.752} C_VEL
LIN {X 0,Y 664.323,Z 1006.994,A -85,B 0,C 180,E1 24540.281,E2 24540.281} C_VEL
LIN {X 0,Y 665.829,Z 984.494,A -85,B 0,C 180,E1 24538.847,E2 24538.847} C_VEL
LIN {X 0,Y 667.184,Z 963.891,A -85,B 0,C 180,E1 24537.699,E2 24537.699} C_VEL
LIN {X 0,Y 668.767,Z 939.295,A -85,B 0,C 180,E1 24536.517,E2 24536.517} C_VEL
LIN {X 0,Y 669.959,Z 918.16,A -85,B 0,C 180,E1 24535.657,E2 24535.657} C_VEL
LIN {X 0,Y 670.95,Z 899.023,A -85,B 0,C 180,E1 24534.989,E2 24534.989} C_VEL
LIN {X 0,Y 671.867,Z 878.988,A -85,B 0,C 180,E1 24534.395,E2 24534.395} C_VEL
LIN {X 0,Y 672.87,Z 853.839,A -85,B 0,C 180,E1 24533.795,E2 24533.795} C_VEL
LIN {X 0,Y 673.523,Z 828.688,A -85,B 0,C 180,E1 24533.363,E2 24533.363} C_VEL
LIN {X 0,Y 676.5,Z 594.686,A -85,B 0,C 180,E1 24530.439,E2 24530.439} C_VEL
LIN {X 0,Y 678.945,Z 420.53,A -85,B 0,C 180,E1 24528.196,E2 24528.196} C_VEL
LIN {X 0,Y 673.507,Z 395.332,A -85,B 0,C 180,E1 24527.36,E2 24527.36} C_VEL
LIN {X 0,Y 675.357,Z 362.566,A -85,B 0,C 180,E1 24525.108,E2 24525.108} C_VEL
LIN {X 0,Y 666.903,Z 343.82,A -85,B 0,C 180,E1 24522.897,E2 24522.897} C_VEL
LIN {X 0,Y 660.416,Z 330.629,A -85,B 0,C 180,E1 24521.194,E2 24521.194} C_VEL
LIN {X 0,Y 658.004,Z 325.952,A -85,B 0,C 180,E1 24520.555,E2 24520.555} C_VEL
LIN {X 0,Y 656.734,Z 322.64,A -85,B 0,C 180,E1 24520.093,E2 24520.093} C_VEL
LIN {X 0,Y 656.66,Z 322.404,A -85,B 0,C 180,E1 24517.072,E2 24517.072} C_VEL
LIN {X 0,Y 656.684,Z 322.41,A -85,B 0,C 180,E1 24514.184,E2 24514.184} C_VEL
LIN {X 0,Y 656.673,Z 322.431,A -85,B 0,C 180,E1 24510.975,E2 24510.975} C_VEL
LIN {X 0,Y 656.702,Z 322.404,A -85,B 0,C 180,E1 24507.967,E2 24507.967} C_VEL
LIN {X 0,Y 656.676,Z 322.415,A -85,B 0,C 180,E1 24504.84,E2 24504.84} C_VEL
LIN {X 0,Y 656.708,Z 322.425,A -85,B 0,C 180,E1 24501.809,E2 24501.809} C_VEL
LIN {X 0,Y 656.684,Z 322.399,A -85,B 0,C 180,E1 24498.726,E2 24498.726} C_VEL
LIN {X 0,Y 656.704,Z 322.432,A -85,B 0,C 180,E1 24495.635,E2 24495.635} C_VEL
LIN {X 0,Y 656.688,Z 322.394,A -85,B 0,C 180,E1 24492.576,E2 24492.576} C_VEL
LIN {X 0,Y 656.7,Z 322.43,A -85,B 0,C 180,E1 24489.553,E2 24489.553} C_VEL
LIN {X 0,Y 656.695,Z 322.392,A -85,B 0,C 180,E1 24486.469,E2 24486.469} C_VEL
LIN {X 0,Y 656.694,Z 322.43,A -85,B 0,C 180,E1 24483.404,E2 24483.404} C_VEL
LIN {X 0,Y 656.7,Z 322.394,A -85,B 0,C 180,E1 24480.349,E2 24480.349} C_VEL
LIN {X 0,Y 656.683,Z 322.432,A -85,B 0,C 180,E1 24477.231,E2 24477.231} C_VEL
LIN {X 0,Y 656.701,Z 322.396,A -85,B 0,C 180,E1 24474.145,E2 24474.145} C_VEL
LIN {X 0,Y 656.677,Z 322.432,A -85,B 0,C 180,E1 24471.153,E2 24471.153} C_VEL
LIN {X 0,Y 656.704,Z 322.397,A -85,B 0,C 180,E1 24468.138,E2 24468.138} C_VEL
LIN {X 0,Y 656.675,Z 322.433,A -85,B 0,C 180,E1 24465.088,E2 24465.088} C_VEL
LIN {X 0,Y 656.695,Z 322.396,A -85,B 0,C 180,E1 24462.087,E2 24462.087} C_VEL
LIN {X 0,Y 656.663,Z 322.43,A -85,B 0,C 180,E1 24458.939,E2 24458.939} C_VEL
LIN {X 0,Y 656.673,Z 322.405,A -85,B 0,C 180,E1 24456.107,E2 24456.107} C_VEL
LIN {X 0,Y 656.659,Z 322.416,A -85,B 0,C 180,E1 24452.917,E2 24452.917} C_VEL
LIN {X 0,Y 656.648,Z 322.431,A -85,B 0,C 180,E1 24450.219,E2 24450.219} C_VEL
LIN {X 0,Y 656.69,Z 322.402,A -85,B 0,C 180,E1 24447.176,E2 24447.176} C_VEL
LIN {X 0,Y 656.629,Z 322.42,A -85,B 0,C 180,E1 24444.404,E2 24444.404} C_VEL
LIN {X 0,Y 656.686,Z 322.475,A -85,B 0,C 180,E1 24441.594,E2 24441.594} C_VEL
LIN {X 0,Y 656.817,Z 323.068,A -85,B 0,C 180,E1 24441.354,E2 24441.354} C_VEL
LIN {X 0,Y 658.418,Z 326.521,A -85,B 0,C 180,E1 24440.896,E2 24440.896} C_VEL
LIN {X 0,Y 665.259,Z 339.982,A -85,B 0,C 180,E1 24439.17,E2 24439.17} C_VEL
LIN {X 0,Y 670.759,Z 350.998,A -85,B 0,C 180,E1 24437.87,E2 24437.87} C_VEL
LIN {X 0,Y 681.552,Z 366.683,A -85,B 0,C 180,E1 24436.668,E2 24436.668} C_VEL
LIN {X 0,Y 683.868,Z 377.867,A -85,B 0,C 180,E1 24436.296,E2 24436.296} C_VEL
LIN {X 0,Y 680.68,Z 590.524,A -85,B 0,C 180,E1 24433.467,E2 24433.467} C_VEL
LIN {X 0,Y 677.581,Z 814.712,A -85,B 0,C 180,E1 24430.576,E2 24430.576} C_VEL
LIN {X 0,Y 676.815,Z 842.535,A -85,B 0,C 180,E1 24430.147,E2 24430.147} C_VEL
LIN {X 0,Y 675.912,Z 866.19,A -85,B 0,C 180,E1 24429.649,E2 24429.649} C_VEL
LIN {X 0,Y 674.704,Z 892.386,A -85,B 0,C 180,E1 24428.945,E2 24428.945} C_VEL
LIN {X 0,Y 673.229,Z 918.738,A -85,B 0,C 180,E1 24428.05,E2 24428.05} C_VEL
LIN {X 0,Y 671.901,Z 939.832,A -85,B 0,C 180,E1 24427.206,E2 24427.206} C_VEL
LIN {X 0,Y 670.502,Z 960.715,A -85,B 0,C 180,E1 24426.247,E2 24426.247} C_VEL
LIN {X 0,Y 668.873,Z 983.896,A -85,B 0,C 180,E1 24425.031,E2 24425.031} C_VEL
LIN {X 0,Y 666.981,Z 1008.529,A -85,B 0,C 180,E1 24423.538,E2 24423.538} C_VEL
LIN {X 0,Y 665.451,Z 1028.179,A -85,B 0,C 180,E1 24422.19,E2 24422.19} C_VEL
LIN {X 0,Y 663.951,Z 1048.29,A -85,B 0,C 180,E1 24420.648,E2 24420.648} C_VEL
LIN {X 0,Y 662.313,Z 1070.05,A -85,B 0,C 180,E1 24418.76,E2 24418.76} C_VEL
LIN {X 0,Y 661.059,Z 1086.85,A -85,B 0,C 180,E1 24417.131,E2 24417.131} C_VEL
LIN {X 0,Y 659.908,Z 1104.462,A -85,B 0,C 180,E1 24415.234,E2 24415.234} C_VEL
LIN {X 0,Y 658.773,Z 1121.892,A -85,B 0,C 180,E1 24413.104,E2 24413.104} C_VEL
LIN {X 0,Y 658.001,Z 1135.752,A -85,B 0,C 180,E1 24411.202,E2 24411.202} C_VEL
LIN {X 0,Y 657.304,Z 1150.03,A -85,B 0,C 180,E1 24408.998,E2 24408.998} C_VEL
LIN {X 0,Y 656.752,Z 1162.678,A -85,B 0,C 180,E1 24406.723,E2 24406.723} C_VEL
LIN {X 0,Y 656.451,Z 1171.896,A -85,B 0,C 180,E1 24404.826,E2 24404.826} C_VEL
LIN {X 0,Y 656.232,Z 1179.871,A -85,B 0,C 180,E1 24402.943,E2 24402.943} C_VEL
LIN {X 0,Y 656.05,Z 1187.892,A -85,B 0,C 180,E1 24400.716,E2 24400.716} C_VEL
LIN {X 0,Y 655.97,Z 1194.694,A -85,B 0,C 180,E1 24398.326,E2 24398.326} C_VEL
LIN {X 0,Y 655.929,Z 1199.41,A -85,B 0,C 180,E1 24396.125,E2 24396.125} C_VEL
LIN {X 0,Y 655.91,Z 1202.789,A -85,B 0,C 180,E1 24393.846,E2 24393.846} C_VEL
LIN {X 0,Y 655.911,Z 1204.624,A -85,B 0,C 180,E1 24391.485,E2 24391.485} C_VEL
LIN {X 0,Y 655.893,Z 1204.849,A -85,B 0,C 180,E1 24389.388,E2 24389.388} C_VEL
LIN {X 0,Y 655.908,Z 1203.947,A -85,B 0,C 180,E1 24387.379,E2 24387.379} C_VEL
LIN {X 0,Y 655.92,Z 1201.427,A -85,B 0,C 180,E1 24385.103,E2 24385.103} C_VEL
LIN {X 0,Y 655.949,Z 1197.151,A -85,B 0,C 180,E1 24382.731,E2 24382.731} C_VEL
LIN {X 0,Y 656.008,Z 1191.375,A -85,B 0,C 180,E1 24380.437,E2 24380.437} C_VEL
LIN {X 0,Y 656.126,Z 1184.277,A -85,B 0,C 180,E1 24378.217,E2 24378.217} C_VEL
LIN {X 0,Y 656.39,Z 1174.089,A -85,B 0,C 180,E1 24375.658,E2 24375.658} C_VEL
LIN {X 0,Y 656.692,Z 1164.276,A -85,B 0,C 180,E1 24373.588,E2 24373.588} C_VEL
LIN {X 0,Y 657.111,Z 1154.138,A -85,B 0,C 180,E1 24371.716,E2 24371.716} C_VEL
LIN {X 0,Y 657.763,Z 1140.776,A -85,B 0,C 180,E1 24369.535,E2 24369.535} C_VEL
LIN {X 0,Y 658.6,Z 1125.099,A -85,B 0,C 180,E1 24367.318,E2 24367.318} C_VEL
LIN {X 0,Y 659.477,Z 1110.397,A -85,B 0,C 180,E1 24365.466,E2 24365.466} C_VEL
LIN {X 0,Y 660.73,Z 1092.314,A -85,B 0,C 180,E1 24363.428,E2 24363.428} C_VEL
LIN {X 0,Y 662.002,Z 1073.81,A -85,B 0,C 180,E1 24361.59,E2 24361.59} C_VEL
LIN {X 0,Y 663.29,Z 1056.832,A -85,B 0,C 180,E1 24360.068,E2 24360.068} C_VEL
LIN {X 0,Y 664.965,Z 1035.518,A -85,B 0,C 180,E1 24358.347,E2 24358.347} C_VEL
LIN {X 0,Y 666.619,Z 1012.989,A -85,B 0,C 180,E1 24356.755,E2 24356.755} C_VEL
LIN {X 0,Y 668.132,Z 993.006,A -85,B 0,C 180,E1 24355.498,E2 24355.498} C_VEL
LIN {X 0,Y 669.921,Z 969.546,A -85,B 0,C 180,E1 24354.192,E2 24354.192} C_VEL
LIN {X 0,Y 671.589,Z 945.096,A -85,B 0,C 180,E1 24353.024,E2 24353.024} C_VEL
LIN {X 0,Y 672.928,Z 923.865,A -85,B 0,C 180,E1 24352.145,E2 24352.145} C_VEL
LIN {X 0,Y 674.048,Z 903.751,A -85,B 0,C 180,E1 24351.422,E2 24351.422} C_VEL
LIN {X 0,Y 675.237,Z 881.05,A -85,B 0,C 180,E1 24350.731,E2 24350.731} C_VEL
LIN {X 0,Y 676.434,Z 854.337,A -85,B 0,C 180,E1 24350.081,E2 24350.081} C_VEL
LIN {X 0,Y 677.27,Z 827.564,A -85,B 0,C 180,E1 24349.604,E2 24349.604} C_VEL
LIN {X 0,Y 680.311,Z 616.305,A -85,B 0,C 180,E1 24346.87,E2 24346.87} C_VEL
LIN {X 0,Y 683.318,Z 412.848,A -85,B 0,C 180,E1 24344.175,E2 24344.175} C_VEL
LIN {X 0,Y 683.741,Z 376.399,A -85,B 0,C 180,E1 24343.671,E2 24343.671} C_VEL
LIN {X 0,Y 681.188,Z 365.954,A -85,B 0,C 180,E1 24343.289,E2 24343.289} C_VEL
LIN {X 0,Y 670.256,Z 350.146,A -85,B 0,C 180,E1 24342.053,E2 24342.053} C_VEL
LIN {X 0,Y 662.397,Z 334.517,A -85,B 0,C 180,E1 24340.133,E2 24340.133} C_VEL
LIN {X 0,Y 660.056,Z 330.061,A -85,B 0,C 180,E1 24339.551,E2 24339.551} C_VEL
LIN {X 0,Y 658.288,Z 326.346,A -85,B 0,C 180,E1 24339.077,E2 24339.077} C_VEL
LIN {X 0,Y 656.731,Z 322.639,A -85,B 0,C 180,E1 24338.566,E2 24338.566} C_VEL
LIN {X 0,Y 656.629,Z 322.418,A -85,B 0,C 180,E1 24335.677,E2 24335.677} C_VEL
LIN {X 0,Y 656.674,Z 322.405,A -85,B 0,C 180,E1 24332.928,E2 24332.928} C_VEL
LIN {X 0,Y 656.652,Z 322.431,A -85,B 0,C 180,E1 24329.863,E2 24329.863} C_VEL
LIN {X 0,Y 656.649,Z 322.416,A -85,B 0,C 180,E1 24327.182,E2 24327.182} C_VEL
LIN {X 0,Y 656.692,Z 322.405,A -85,B 0,C 180,E1 24324.083,E2 24324.083} C_VEL
LIN {X 0,Y 656.656,Z 322.43,A -85,B 0,C 180,E1 24321.154,E2 24321.154} C_VEL
LIN {X 0,Y 656.705,Z 322.396,A -85,B 0,C 180,E1 24318.096,E2 24318.096} C_VEL
LIN {X 0,Y 656.661,Z 322.432,A -85,B 0,C 180,E1 24315.093,E2 24315.093} C_VEL
LIN {X 0,Y 656.704,Z 322.396,A -85,B 0,C 180,E1 24312.129,E2 24312.129} C_VEL
LIN {X 0,Y 656.668,Z 322.429,A -85,B 0,C 180,E1 24309.112,E2 24309.112} C_VEL
LIN {X 0,Y 656.699,Z 322.396,A -85,B 0,C 180,E1 24306.118,E2 24306.118} C_VEL
LIN {X 0,Y 656.676,Z 322.429,A -85,B 0,C 180,E1 24303.055,E2 24303.055} C_VEL
LIN {X 0,Y 656.696,Z 322.395,A -85,B 0,C 180,E1 24300.087,E2 24300.087} C_VEL
LIN {X 0,Y 656.685,Z 322.425,A -85,B 0,C 180,E1 24297.032,E2 24297.032} C_VEL
LIN {X 0,Y 656.694,Z 322.394,A -85,B 0,C 180,E1 24293.969,E2 24293.969} C_VEL
LIN {X 0,Y 656.69,Z 322.423,A -85,B 0,C 180,E1 24290.889,E2 24290.889} C_VEL
LIN {X 0,Y 656.687,Z 322.395,A -85,B 0,C 180,E1 24287.828,E2 24287.828} C_VEL
LIN {X 0,Y 656.697,Z 322.425,A -85,B 0,C 180,E1 24284.818,E2 24284.818} C_VEL
LIN {X 0,Y 656.686,Z 322.399,A -85,B 0,C 180,E1 24281.812,E2 24281.812} C_VEL
LIN {X 0,Y 656.704,Z 322.427,A -85,B 0,C 180,E1 24278.719,E2 24278.719} C_VEL
LIN {X 0,Y 656.676,Z 322.406,A -85,B 0,C 180,E1 24275.629,E2 24275.629} C_VEL
LIN {X 0,Y 656.706,Z 322.422,A -85,B 0,C 180,E1 24272.58,E2 24272.58} C_VEL
LIN {X 0,Y 656.672,Z 322.428,A -85,B 0,C 180,E1 24269.521,E2 24269.521} C_VEL
LIN {X 0,Y 656.703,Z 322.398,A -85,B 0,C 180,E1 24266.55,E2 24266.55} C_VEL
LIN {X 0,Y 656.666,Z 322.413,A -85,B 0,C 180,E1 24263.461,E2 24263.461} C_VEL
LIN {X 0,Y 656.692,Z 322.429,A -85,B 0,C 180,E1 24260.538,E2 24260.538} C_VEL
LIN {X 0,Y 656.414,Z 323.165,A -85,B 0,C 180,E1 24260.224,E2 24260.224} C_VEL
LIN {X 0,Y 655.276,Z 326.358,A -85,B 0,C 180,E1 24259.785,E2 24259.785} C_VEL
LIN {X 0,Y 654.019,Z 332.911,A -85,B 0,C 180,E1 24259.2,E2 24259.2} C_VEL
LIN {X 0,Y 654.587,Z 335.796,A -85,B 0,C 180,E1 24258.883,E2 24258.883} C_VEL
LIN {X 0,Y 654.814,Z 336.179,A -85,B 0,C 180,E1 24258.827,E2 24258.827} C_VEL
LIN {X 0,Y 663.221,Z 353.834,A -85,B 0,C 180,E1 24256.569,E2 24256.569} C_VEL
LIN {X 0,Y 668.953,Z 366.766,A -85,B 0,C 180,E1 24255.045,E2 24255.045} C_VEL
LIN {X 0,Y 667.234,Z 395.296,A -85,B 0,C 180,E1 24253.074,E2 24253.074} C_VEL
LIN {X 0,Y 673.21,Z 423.154,A -85,B 0,C 180,E1 24252.152,E2 24252.152} C_VEL
LIN {X 0,Y 669.464,Z 657.556,A -85,B 0,C 180,E1 24249.112,E2 24249.112} C_VEL
LIN {X 0,Y 667.069,Z 830.476,A -85,B 0,C 180,E1 24246.931,E2 24246.931} C_VEL
LIN {X 0,Y 666.24,Z 857.351,A -85,B 0,C 180,E1 24246.447,E2 24246.447} C_VEL
LIN {X 0,Y 665.255,Z 880.091,A -85,B 0,C 180,E1 24245.889,E2 24245.889} C_VEL
LIN {X 0,Y 664.297,Z 899.424,A -85,B 0,C 180,E1 24245.309,E2 24245.309} C_VEL
LIN {X 0,Y 663.228,Z 918.483,A -85,B 0,C 180,E1 24244.636,E2 24244.636} C_VEL
LIN {X 0,Y 661.816,Z 941.794,A -85,B 0,C 180,E1 24243.674,E2 24243.674} C_VEL
LIN {X 0,Y 660.157,Z 965.112,A -85,B 0,C 180,E1 24242.526,E2 24242.526} C_VEL
LIN {X 0,Y 658.706,Z 985.466,A -85,B 0,C 180,E1 24241.376,E2 24241.376} C_VEL
LIN {X 0,Y 656.975,Z 1008.966,A -85,B 0,C 180,E1 24239.846,E2 24239.846} C_VEL
LIN {X 0,Y 655.549,Z 1027.552,A -85,B 0,C 180,E1 24238.466,E2 24238.466} C_VEL
LIN {X 0,Y 654.091,Z 1047.494,A -85,B 0,C 180,E1 24236.805,E2 24236.805} C_VEL
LIN {X 0,Y 652.717,Z 1066.235,A -85,B 0,C 180,E1 24235.011,E2 24235.011} C_VEL
LIN {X 0,Y 651.628,Z 1082.048,A -85,B 0,C 180,E1 24233.321,E2 24233.321} C_VEL
LIN {X 0,Y 650.558,Z 1098.957,A -85,B 0,C 180,E1 24231.268,E2 24231.268} C_VEL
LIN {X 0,Y 649.836,Z 1111.757,A -85,B 0,C 180,E1 24229.505,E2 24229.505} C_VEL
LIN {X 0,Y 649.177,Z 1125.392,A -85,B 0,C 180,E1 24227.386,E2 24227.386} C_VEL
LIN {X 0,Y 648.677,Z 1136.922,A -85,B 0,C 180,E1 24225.283,E2 24225.283} C_VEL
LIN {X 0,Y 648.365,Z 1145.995,A -85,B 0,C 180,E1 24223.375,E2 24223.375} C_VEL
LIN {X 0,Y 648.121,Z 1155.094,A -85,B 0,C 180,E1 24221.119,E2 24221.119} C_VEL
LIN {X 0,Y 648.015,Z 1161.756,A -85,B 0,C 180,E1 24219.055,E2 24219.055} C_VEL
LIN {X 0,Y 647.948,Z 1166.637,A -85,B 0,C 180,E1 24217.181,E2 24217.181} C_VEL
LIN {X 0,Y 647.918,Z 1170.544,A -85,B 0,C 180,E1 24215.224,E2 24215.224} C_VEL
LIN {X 0,Y 647.903,Z 1173.631,A -85,B 0,C 180,E1 24212.831,E2 24212.831} C_VEL
LIN {X 0,Y 647.905,Z 1174.77,A -85,B 0,C 180,E1 24210.884,E2 24210.884} C_VEL
LIN {X 0,Y 647.909,Z 1174.77,A -85,B 0,C 180,E1 24209.028,E2 24209.028} C_VEL
LIN {X 0,Y 647.909,Z 1173.499,A -85,B 0,C 180,E1 24206.904,E2 24206.904} C_VEL
LIN {X 0,Y 647.916,Z 1170.385,A -85,B 0,C 180,E1 24204.599,E2 24204.599} C_VEL
LIN {X 0,Y 647.951,Z 1166.639,A -85,B 0,C 180,E1 24202.731,E2 24202.731} C_VEL
LIN {X 0,Y 648.015,Z 1161.759,A -85,B 0,C 180,E1 24200.856,E2 24200.856} C_VEL
LIN {X 0,Y 648.147,Z 1154.46,A -85,B 0,C 180,E1 24198.612,E2 24198.612} C_VEL
LIN {X 0,Y 648.383,Z 1145.588,A -85,B 0,C 180,E1 24196.444,E2 24196.444} C_VEL
LIN {X 0,Y 648.673,Z 1136.914,A -85,B 0,C 180,E1 24194.626,E2 24194.626} C_VEL
LIN {X 0,Y 649.172,Z 1125.38,A -85,B 0,C 180,E1 24192.522,E2 24192.522} C_VEL
LIN {X 0,Y 649.833,Z 1111.737,A -85,B 0,C 180,E1 24190.402,E2 24190.402} C_VEL
LIN {X 0,Y 650.609,Z 1098.217,A -85,B 0,C 180,E1 24188.545,E2 24188.545} C_VEL
LIN {X 0,Y 651.674,Z 1081.155,A -85,B 0,C 180,E1 24186.489,E2 24186.489} C_VEL
LIN {X 0,Y 652.736,Z 1065.923,A -85,B 0,C 180,E1 24184.867,E2 24184.867} C_VEL
LIN {X 0,Y 654.104,Z 1047.413,A -85,B 0,C 180,E1 24183.098,E2 24183.098} C_VEL
LIN {X 0,Y 655.55,Z 1027.509,A -85,B 0,C 180,E1 24181.44,E2 24181.44} C_VEL
LIN {X 0,Y 656.986,Z 1008.834,A -85,B 0,C 180,E1 24180.054,E2 24180.054} C_VEL
LIN {X 0,Y 658.716,Z 985.292,A -85,B 0,C 180,E1 24178.523,E2 24178.523} C_VEL
LIN {X 0,Y 660.192,Z 964.694,A -85,B 0,C 180,E1 24177.362,E2 24177.362} C_VEL
LIN {X 0,Y 661.878,Z 940.741,A -85,B 0,C 180,E1 24176.189,E2 24176.189} C_VEL
LIN {X 0,Y 663.271,Z 917.737,A -85,B 0,C 180,E1 24175.245,E2 24175.245} C_VEL
LIN {X 0,Y 664.36,Z 898.26,A -85,B 0,C 180,E1 24174.563,E2 24174.563} C_VEL
LIN {X 0,Y 665.347,Z 878.234,A -85,B 0,C 180,E1 24173.97,E2 24173.97} C_VEL
LIN {X 0,Y 666.406,Z 852.766,A -85,B 0,C 180,E1 24173.365,E2 24173.365} C_VEL
LIN {X 0,Y 667.1,Z 828.323,A -85,B 0,C 180,E1 24172.947,E2 24172.947} C_VEL
LIN {X 0,Y 670.464,Z 588.246,A -85,B 0,C 180,E1 24169.916,E2 24169.916} C_VEL
LIN {X 0,Y 673.12,Z 422.238,A -85,B 0,C 180,E1 24167.737,E2 24167.737} C_VEL
LIN {X 0,Y 667.211,Z 394.691,A -85,B 0,C 180,E1 24166.803,E2 24166.803} C_VEL
LIN {X 0,Y 668.838,Z 366.309,A -85,B 0,C 180,E1 24164.82,E2 24164.82} C_VEL
LIN {X 0,Y 660.554,Z 348.195,A -85,B 0,C 180,E1 24162.638,E2 24162.638} C_VEL
LIN {X 0,Y 654.453,Z 335.63,A -85,B 0,C 180,E1 24160.998,E2 24160.998} C_VEL
LIN {X 0,Y 650.425,Z 327.37,A -85,B 0,C 180,E1 24159.87,E2 24159.87} C_VEL
LIN {X 0,Y 648.763,Z 323.618,A -85,B 0,C 180,E1 24159.314,E2 24159.314} C_VEL
LIN {X 0,Y 648.716,Z 323.398,A -85,B 0,C 180,E1 24156.58,E2 24156.58} C_VEL
LIN {X 0,Y 648.766,Z 323.385,A -85,B 0,C 180,E1 24153.488,E2 24153.488} C_VEL
LIN {X 0,Y 648.728,Z 323.418,A -85,B 0,C 180,E1 24150.47,E2 24150.47} C_VEL
LIN {X 0,Y 648.77,Z 323.405,A -85,B 0,C 180,E1 24147.412,E2 24147.412} C_VEL
LIN {X 0,Y 648.731,Z 323.393,A -85,B 0,C 180,E1 24144.371,E2 24144.371} C_VEL
LIN {X 0,Y 648.766,Z 323.417,A -85,B 0,C 180,E1 24141.329,E2 24141.329} C_VEL
LIN {X 0,Y 648.74,Z 323.385,A -85,B 0,C 180,E1 24138.233,E2 24138.233} C_VEL
LIN {X 0,Y 648.76,Z 323.415,A -85,B 0,C 180,E1 24135.189,E2 24135.189} C_VEL
LIN {X 0,Y 648.746,Z 323.383,A -85,B 0,C 180,E1 24132.1,E2 24132.1} C_VEL
LIN {X 0,Y 648.756,Z 323.412,A -85,B 0,C 180,E1 24129.045,E2 24129.045} C_VEL
LIN {X 0,Y 648.754,Z 323.381,A -85,B 0,C 180,E1 24125.927,E2 24125.927} C_VEL
LIN {X 0,Y 648.755,Z 323.413,A -85,B 0,C 180,E1 24122.827,E2 24122.827} C_VEL
LIN {X 0,Y 648.765,Z 323.382,A -85,B 0,C 180,E1 24119.647,E2 24119.647} C_VEL
LIN {X 0,Y 648.763,Z 323.414,A -85,B 0,C 180,E1 24116.466,E2 24116.466} C_VEL
LIN {X 0,Y 648.741,Z 323.388,A -85,B 0,C 180,E1 24113.273,E2 24113.273} C_VEL
LIN {X 0,Y 648.766,Z 323.413,A -85,B 0,C 180,E1 24110.239,E2 24110.239} C_VEL
LIN {X 0,Y 648.732,Z 323.393,A -85,B 0,C 180,E1 24107.086,E2 24107.086} C_VEL
LIN {X 0,Y 648.766,Z 323.415,A -85,B 0,C 180,E1 24104.077,E2 24104.077} C_VEL
LIN {X 0,Y 648.723,Z 323.402,A -85,B 0,C 180,E1 24100.928,E2 24100.928} C_VEL
LIN {X 0,Y 648.754,Z 323.405,A -85,B 0,C 180,E1 24098.005,E2 24098.005} C_VEL
LIN {X 0,Y 648.722,Z 323.419,A -85,B 0,C 180,E1 24094.921,E2 24094.921} C_VEL
LIN {X 0,Y 648.716,Z 323.393,A -85,B 0,C 180,E1 24092.158,E2 24092.158} C_VEL
LIN {X 0,Y 648.723,Z 323.415,A -85,B 0,C 180,E1 24088.913,E2 24088.913} C_VEL
LIN {X 0,Y 648.7,Z 323.411,A -85,B 0,C 180,E1 24086.18,E2 24086.18} C_VEL
LIN {X 0,Y 648.746,Z 323.387,A -85,B 0,C 180,E1 24083.121,E2 24083.121} C_VEL
LIN {X 0,Y 648.735,Z 323.727,A -85,B 0,C 180,E1 24082.192,E2 24082.192} C_VEL
LIN {X 0,Y 650.254,Z 327.219,A -85,B 0,C 180,E1 24081.706,E2 24081.706} C_VEL
LIN {X 0,Y 651.32,Z 329.038,A -85,B 0,C 180,E1 24081.444,E2 24081.444} C_VEL
LIN {X 0,Y 659.698,Z 345.755,A -85,B 0,C 180,E1 24079.273,E2 24079.273} C_VEL
LIN {X 0,Y 662.719,Z 351.694,A -85,B 0,C 180,E1 24078.574,E2 24078.574} C_VEL
LIN {X 0,Y 676.597,Z 371.426,A -85,B 0,C 180,E1 24077.042,E2 24077.042} C_VEL
LIN {X 0,Y 678.299,Z 379.932,A -85,B 0,C 180,E1 24076.759,E2 24076.759} C_VEL
LIN {X 0,Y 674.849,Z 591.878,A -85,B 0,C 180,E1 24073.919,E2 24073.919} C_VEL
LIN {X 0,Y 671.483,Z 815.8,A -85,B 0,C 180,E1 24071.008,E2 24071.008} C_VEL
LIN {X 0,Y 670.668,Z 842.835,A -85,B 0,C 180,E1 24070.585,E2 24070.585} C_VEL
LIN {X 0,Y 669.712,Z 866.17,A -85,B 0,C 180,E1 24070.09,E2 24070.09} C_VEL
LIN {X 0,Y 668.437,Z 891.872,A -85,B 0,C 180,E1 24069.398,E2 24069.398} C_VEL
LIN {X 0,Y 666.805,Z 918.734,A -85,B 0,C 180,E1 24068.484,E2 24068.484} C_VEL
LIN {X 0,Y 665.363,Z 939.923,A -85,B 0,C 180,E1 24067.63,E2 24067.63} C_VEL
LIN {X 0,Y 663.855,Z 960.711,A -85,B 0,C 180,E1 24066.669,E2 24066.669} C_VEL
LIN {X 0,Y 662.098,Z 983.899,A -85,B 0,C 180,E1 24065.443,E2 24065.443} C_VEL
LIN {X 0,Y 660.055,Z 1008.598,A -85,B 0,C 180,E1 24063.932,E2 24063.932} C_VEL
LIN {X 0,Y 658.45,Z 1027.575,A -85,B 0,C 180,E1 24062.621,E2 24062.621} C_VEL
LIN {X 0,Y 656.824,Z 1047.081,A -85,B 0,C 180,E1 24061.119,E2 24061.119} C_VEL
LIN {X 0,Y 654.984,Z 1069.754,A -85,B 0,C 180,E1 24059.142,E2 24059.142} C_VEL
LIN {X 0,Y 653.645,Z 1086.385,A -85,B 0,C 180,E1 24057.514,E2 24057.514} C_VEL
LIN {X 0,Y 652.37,Z 1103.305,A -85,B 0,C 180,E1 24055.679,E2 24055.679} C_VEL
LIN {X 0,Y 651.105,Z 1121.563,A -85,B 0,C 180,E1 24053.437,E2 24053.437} C_VEL
LIN {X 0,Y 650.244,Z 1135.43,A -85,B 0,C 180,E1 24051.515,E2 24051.515} C_VEL
LIN {X 0,Y 649.486,Z 1149.55,A -85,B 0,C 180,E1 24049.313,E2 24049.313} C_VEL
LIN {X 0,Y 648.875,Z 1162.214,A -85,B 0,C 180,E1 24047.024,E2 24047.024} C_VEL
LIN {X 0,Y 648.513,Z 1171.487,A -85,B 0,C 180,E1 24045.103,E2 24045.103} C_VEL
LIN {X 0,Y 648.28,Z 1179.515,A -85,B 0,C 180,E1 24043.195,E2 24043.195} C_VEL
LIN {X 0,Y 648.084,Z 1187.034,A -85,B 0,C 180,E1 24041.112,E2 24041.112} C_VEL
LIN {X 0,Y 647.987,Z 1193.816,A -85,B 0,C 180,E1 24038.787,E2 24038.787} C_VEL
LIN {X 0,Y 647.935,Z 1199.101,A -85,B 0,C 180,E1 24036.371,E2 24036.371} C_VEL
LIN {X 0,Y 647.918,Z 1202.476,A -85,B 0,C 180,E1 24034.159,E2 24034.159} C_VEL
LIN {X 0,Y 647.907,Z 1204.549,A -85,B 0,C 180,E1 24031.769,E2 24031.769} C_VEL
LIN {X 0,Y 647.892,Z 1204.872,A -85,B 0,C 180,E1 24029.469,E2 24029.469} C_VEL
LIN {X 0,Y 647.909,Z 1203.944,A -85,B 0,C 180,E1 24027.346,E2 24027.346} C_VEL
LIN {X 0,Y 647.922,Z 1201.427,A -85,B 0,C 180,E1 24025.042,E2 24025.042} C_VEL
LIN {X 0,Y 647.951,Z 1197.151,A -85,B 0,C 180,E1 24022.641,E2 24022.641} C_VEL
LIN {X 0,Y 648.018,Z 1191.372,A -85,B 0,C 180,E1 24020.318,E2 24020.318} C_VEL
LIN {X 0,Y 648.146,Z 1184.277,A -85,B 0,C 180,E1 24018.07,E2 24018.07} C_VEL
LIN {X 0,Y 648.438,Z 1174.335,A -85,B 0,C 180,E1 24015.534,E2 24015.534} C_VEL
LIN {X 0,Y 648.77,Z 1164.541,A -85,B 0,C 180,E1 24013.434,E2 24013.434} C_VEL
LIN {X 0,Y 649.237,Z 1154.234,A -85,B 0,C 180,E1 24011.503,E2 24011.503} C_VEL
LIN {X 0,Y 649.925,Z 1141.36,A -85,B 0,C 180,E1 24009.371,E2 24009.371} C_VEL
LIN {X 0,Y 650.838,Z 1125.797,A -85,B 0,C 180,E1 24007.127,E2 24007.127} C_VEL
LIN {X 0,Y 651.805,Z 1111.148,A -85,B 0,C 180,E1 24005.251,E2 24005.251} C_VEL
LIN {X 0,Y 653.114,Z 1093.72,A -85,B 0,C 180,E1 24003.25,E2 24003.25} C_VEL
LIN {X 0,Y 654.549,Z 1074.823,A -85,B 0,C 180,E1 24001.337,E2 24001.337} C_VEL
LIN {X 0,Y 655.938,Z 1057.941,A -85,B 0,C 180,E1 23999.799,E2 23999.799} C_VEL
LIN {X 0,Y 657.513,Z 1039.183,A -85,B 0,C 180,E1 23998.253,E2 23998.253} C_VEL
LIN {X 0,Y 659.486,Z 1015.133,A -85,B 0,C 180,E1 23996.501,E2 23996.501} C_VEL
LIN {X 0,Y 661.141,Z 994.954,A -85,B 0,C 180,E1 23995.207,E2 23995.207} C_VEL
LIN {X 0,Y 662.831,Z 974.042,A -85,B 0,C 180,E1 23994.016,E2 23994.016} C_VEL
LIN {X 0,Y 664.823,Z 948.452,A -85,B 0,C 180,E1 23992.746,E2 23992.746} C_VEL
LIN {X 0,Y 666.409,Z 925.146,A -85,B 0,C 180,E1 23991.763,E2 23991.763} C_VEL
LIN {X 0,Y 667.661,Z 904.466,A -85,B 0,C 180,E1 23991.01,E2 23991.01} C_VEL
LIN {X 0,Y 668.913,Z 882.27,A -85,B 0,C 180,E1 23990.326,E2 23990.326} C_VEL
LIN {X 0,Y 670.163,Z 856.634,A -85,B 0,C 180,E1 23989.688,E2 23989.688} C_VEL
LIN {X 0,Y 671.135,Z 828.996,A -85,B 0,C 180,E1 23989.181,E2 23989.181} C_VEL
LIN {X 0,Y 673.11,Z 705.184,A -85,B 0,C 180,E1 23987.564,E2 23987.564} C_VEL
LIN {X 0,Y 676.521,Z 487.157,A -85,B 0,C 180,E1 23984.689,E2 23984.689} C_VEL
LIN {X 0,Y 678.164,Z 378.464,A -85,B 0,C 180,E1 23983.207,E2 23983.207} C_VEL
LIN {X 0,Y 676.307,Z 370.867,A -85,B 0,C 180,E1 23982.923,E2 23982.923} C_VEL
LIN {X 0,Y 662.196,Z 350.785,A -85,B 0,C 180,E1 23981.347,E2 23981.347} C_VEL
LIN {X 0,Y 655.024,Z 336.423,A -85,B 0,C 180,E1 23979.535,E2 23979.535} C_VEL
LIN {X 0,Y 650.654,Z 327.723,A -85,B 0,C 180,E1 23978.378,E2 23978.378} C_VEL
LIN {X 0,Y 648.904,Z 324.498,A -85,B 0,C 180,E1 23977.915,E2 23977.915} C_VEL
LIN {X 0,Y 648.703,Z 323.543,A -85,B 0,C 180,E1 23977.729,E2 23977.729} C_VEL
LIN {X 0,Y 648.721,Z 323.418,A -85,B 0,C 180,E1 23975.072,E2 23975.072} C_VEL
LIN {X 0,Y 648.709,Z 323.4,A -85,B 0,C 180,E1 23971.917,E2 23971.917} C_VEL
LIN {X 0,Y 648.707,Z 323.406,A -85,B 0,C 180,E1 23969.249,E2 23969.249} C_VEL
LIN {X 0,Y 648.757,Z 323.42,A -85,B 0,C 180,E1 23966.155,E2 23966.155} C_VEL
LIN {X 0,Y 648.709,Z 323.39,A -85,B 0,C 180,E1 23963.24,E2 23963.24} C_VEL
LIN {X 0,Y 648.772,Z 323.415,A -85,B 0,C 180,E1 23960.29,E2 23960.29} C_VEL
LIN {X 0,Y 648.716,Z 323.393,A -85,B 0,C 180,E1 23957.306,E2 23957.306} C_VEL
LIN {X 0,Y 648.771,Z 323.411,A -85,B 0,C 180,E1 23954.367,E2 23954.367} C_VEL
LIN {X 0,Y 648.727,Z 323.395,A -85,B 0,C 180,E1 23951.288,E2 23951.288} C_VEL
LIN {X 0,Y 648.767,Z 323.41,A -85,B 0,C 180,E1 23948.33,E2 23948.33} C_VEL
LIN {X 0,Y 648.735,Z 323.394,A -85,B 0,C 180,E1 23945.217,E2 23945.217} C_VEL
LIN {X 0,Y 648.765,Z 323.412,A -85,B 0,C 180,E1 23942.208,E2 23942.208} C_VEL
LIN {X 0,Y 648.743,Z 323.387,A -85,B 0,C 180,E1 23939.117,E2 23939.117} C_VEL
LIN {X 0,Y 648.763,Z 323.414,A -85,B 0,C 180,E1 23936.112,E2 23936.112} C_VEL
LIN {X 0,Y 648.749,Z 323.381,A -85,B 0,C 180,E1 23933.006,E2 23933.006} C_VEL
LIN {X 0,Y 648.756,Z 323.414,A -85,B 0,C 180,E1 23929.97,E2 23929.97} C_VEL
LIN {X 0,Y 648.756,Z 323.382,A -85,B 0,C 180,E1 23926.905,E2 23926.905} C_VEL
LIN {X 0,Y 648.754,Z 323.415,A -85,B 0,C 180,E1 23923.893,E2 23923.893} C_VEL
LIN {X 0,Y 648.76,Z 323.39,A -85,B 0,C 180,E1 23920.742,E2 23920.742} C_VEL
LIN {X 0,Y 648.744,Z 323.408,A -85,B 0,C 180,E1 23917.719,E2 23917.719} C_VEL
LIN {X 0,Y 648.767,Z 323.405,A -85,B 0,C 180,E1 23914.63,E2 23914.63} C_VEL
LIN {X 0,Y 648.733,Z 323.388,A -85,B 0,C 180,E1 23911.558,E2 23911.558} C_VEL
LIN {X 0,Y 648.772,Z 323.419,A -85,B 0,C 180,E1 23908.502,E2 23908.502} C_VEL
LIN {X 0,Y 648.726,Z 323.407,A -85,B 0,C 180,E1 23905.392,E2 23905.392} C_VEL
LIN {X 0,Y 648.766,Z 323.385,A -85,B 0,C 180,E1 23902.387,E2 23902.387} C_VEL
LIN {X 0,Y 648.781,Z 323.653,A -85,B 0,C 180,E1 23900.582,E2 23900.582} C_VEL
LIN {X 0,Y 650.117,Z 326.944,A -85,B 0,C 180,E1 23900.107,E2 23900.107} C_VEL
LIN {X 0,Y 651.141,Z 328.79,A -85,B 0,C 180,E1 23899.838,E2 23899.838} C_VEL
LIN {X 0,Y 654.814,Z 336.179,A -85,B 0,C 180,E1 23898.827,E2 23898.827} C_VEL
LIN {X 0,Y 655.56,Z 338.895,A -85,B 0,C 180,E1 23898.525,E2 23898.525} C_VEL
LIN {X 0,Y 654.924,Z 344.771,A -85,B 0,C 180,E1 23898.104,E2 23898.104} C_VEL
LIN {X 0,Y 654.205,Z 350.758,A -85,B 0,C 180,E1 23897.685,E2 23897.685} C_VEL
LIN {X 0,Y 654.855,Z 353.64,A -85,B 0,C 180,E1 23897.387,E2 23897.387} C_VEL
LIN {X 0,Y 662.557,Z 370.886,A -85,B 0,C 180,E1 23895.3,E2 23895.3} C_VEL
LIN {X 0,Y 661.061,Z 395.295,A -85,B 0,C 180,E1 23893.611,E2 23893.611} C_VEL
LIN {X 0,Y 667.463,Z 424.968,A -85,B 0,C 180,E1 23892.611,E2 23892.611} C_VEL
LIN {X 0,Y 663.353,Z 659.711,A -85,B 0,C 180,E1 23889.536,E2 23889.536} C_VEL
LIN {X 0,Y 660.658,Z 831.161,A -85,B 0,C 180,E1 23887.34,E2 23887.34} C_VEL
LIN {X 0,Y 659.746,Z 858.091,A -85,B 0,C 180,E1 23886.846,E2 23886.846} C_VEL
LIN {X 0,Y 658.733,Z 879.997,A -85,B 0,C 180,E1 23886.304,E2 23886.304} C_VEL
LIN {X 0,Y 657.697,Z 899.44,A -85,B 0,C 180,E1 23885.717,E2 23885.717} C_VEL
LIN {X 0,Y 656.467,Z 919.907,A -85,B 0,C 180,E1 23884.986,E2 23884.986} C_VEL
LIN {X 0,Y 654.778,Z 944.841,A -85,B 0,C 180,E1 23883.927,E2 23883.927} C_VEL
LIN {X 0,Y 653.179,Z 966.02,A -85,B 0,C 180,E1 23882.865,E2 23882.865} C_VEL
LIN {X 0,Y 651.559,Z 987.087,A -85,B 0,C 180,E1 23881.657,E2 23881.657} C_VEL
LIN {X 0,Y 649.705,Z 1010.128,A -85,B 0,C 180,E1 23880.127,E2 23880.127} C_VEL
LIN {X 0,Y 648.217,Z 1028.166,A -85,B 0,C 180,E1 23878.768,E2 23878.768} C_VEL
LIN {X 0,Y 646.65,Z 1047.782,A -85,B 0,C 180,E1 23877.112,E2 23877.112} C_VEL
LIN {X 0,Y 645.178,Z 1066.24,A -85,B 0,C 180,E1 23875.324,E2 23875.324} C_VEL
LIN {X 0,Y 643.988,Z 1082.051,A -85,B 0,C 180,E1 23873.615,E2 23873.615} C_VEL
LIN {X 0,Y 642.833,Z 1098.963,A -85,B 0,C 180,E1 23871.536,E2 23871.536} C_VEL
LIN {X 0,Y 642.03,Z 1111.759,A -85,B 0,C 180,E1 23869.752,E2 23869.752} C_VEL
LIN {X 0,Y 641.304,Z 1125.397,A -85,B 0,C 180,E1 23867.606,E2 23867.606} C_VEL
LIN {X 0,Y 640.759,Z 1136.927,A -85,B 0,C 180,E1 23865.476,E2 23865.476} C_VEL
LIN {X 0,Y 640.433,Z 1145.592,A -85,B 0,C 180,E1 23863.636,E2 23863.636} C_VEL
LIN {X 0,Y 640.177,Z 1154.459,A -85,B 0,C 180,E1 23861.441,E2 23861.441} C_VEL
LIN {X 0,Y 640.026,Z 1161.758,A -85,B 0,C 180,E1 23859.169,E2 23859.169} C_VEL
LIN {X 0,Y 639.956,Z 1166.638,A -85,B 0,C 180,E1 23857.271,E2 23857.271} C_VEL
LIN {X 0,Y 639.917,Z 1170.545,A -85,B 0,C 180,E1 23855.29,E2 23855.29} C_VEL
LIN {X 0,Y 639.903,Z 1173.631,A -85,B 0,C 180,E1 23852.866,E2 23852.866} C_VEL
LIN {X 0,Y 639.905,Z 1174.77,A -85,B 0,C 180,E1 23850.895,E2 23850.895} C_VEL
LIN {X 0,Y 639.909,Z 1174.77,A -85,B 0,C 180,E1 23849.015,E2 23849.015} C_VEL
LIN {X 0,Y 639.908,Z 1173.566,A -85,B 0,C 180,E1 23846.955,E2 23846.955} C_VEL
LIN {X 0,Y 639.914,Z 1170.384,A -85,B 0,C 180,E1 23844.531,E2 23844.531} C_VEL
LIN {X 0,Y 639.954,Z 1166.638,A -85,B 0,C 180,E1 23842.639,E2 23842.639} C_VEL
LIN {X 0,Y 640.028,Z 1161.758,A -85,B 0,C 180,E1 23840.74,E2 23840.74} C_VEL
LIN {X 0,Y 640.18,Z 1154.457,A -85,B 0,C 180,E1 23838.468,E2 23838.468} C_VEL
LIN {X 0,Y 640.437,Z 1145.585,A -85,B 0,C 180,E1 23836.272,E2 23836.272} C_VEL
LIN {X 0,Y 640.757,Z 1136.913,A -85,B 0,C 180,E1 23834.431,E2 23834.431} C_VEL
LIN {X 0,Y 641.301,Z 1125.366,A -85,B 0,C 180,E1 23832.298,E2 23832.298} C_VEL
LIN {X 0,Y 642.026,Z 1111.731,A -85,B 0,C 180,E1 23830.153,E2 23830.153} C_VEL
LIN {X 0,Y 642.89,Z 1098.214,A -85,B 0,C 180,E1 23828.275,E2 23828.275} C_VEL
LIN {X 0,Y 644.05,Z 1081.148,A -85,B 0,C 180,E1 23826.194,E2 23826.194} C_VEL
LIN {X 0,Y 645.224,Z 1065.631,A -85,B 0,C 180,E1 23824.523,E2 23824.523} C_VEL
LIN {X 0,Y 646.69,Z 1047.3,A -85,B 0,C 180,E1 23822.754,E2 23822.754} C_VEL
LIN {X 0,Y 648.276,Z 1027.438,A -85,B 0,C 180,E1 23821.084,E2 23821.084} C_VEL
LIN {X 0,Y 649.825,Z 1008.698,A -85,B 0,C 180,E1 23819.68,E2 23819.68} C_VEL
LIN {X 0,Y 651.683,Z 985.278,A -85,B 0,C 180,E1 23818.143,E2 23818.143} C_VEL
LIN {X 0,Y 653.274,Z 964.876,A -85,B 0,C 180,E1 23816.984,E2 23816.984} C_VEL
LIN {X 0,Y 655.054,Z 941.497,A -85,B 0,C 180,E1 23815.825,E2 23815.825} C_VEL
LIN {X 0,Y 656.57,Z 918.12,A -85,B 0,C 180,E1 23814.855,E2 23814.855} C_VEL
LIN {X 0,Y 657.765,Z 898.237,A -85,B 0,C 180,E1 23814.153,E2 23814.153} C_VEL
LIN {X 0,Y 658.837,Z 878.028,A -85,B 0,C 180,E1 23813.551,E2 23813.551} C_VEL
LIN {X 0,Y 659.962,Z 852.494,A -85,B 0,C 180,E1 23812.943,E2 23812.943} C_VEL
LIN {X 0,Y 660.711,Z 828.172,A -85,B 0,C 180,E1 23812.526,E2 23812.526} C_VEL
LIN {X 0,Y 664.391,Z 601.239,A -85,B 0,C 180,E1 23809.613,E2 23809.613} C_VEL
LIN {X 0,Y 667.385,Z 424.222,A -85,B 0,C 180,E1 23807.281,E2 23807.281} C_VEL
LIN {X 0,Y 660.978,Z 394.557,A -85,B 0,C 180,E1 23806.266,E2 23806.266} C_VEL
LIN {X 0,Y 662.467,Z 370.468,A -85,B 0,C 180,E1 23804.57,E2 23804.57} C_VEL
LIN {X 0,Y 654.587,Z 353.17,A -85,B 0,C 180,E1 23802.458,E2 23802.458} C_VEL
LIN {X 0,Y 648.525,Z 340.608,A -85,B 0,C 180,E1 23800.799,E2 23800.799} C_VEL
LIN {X 0,Y 644.356,Z 332.203,A -85,B 0,C 180,E1 23799.626,E2 23799.626} C_VEL
LIN {X 0,Y 642.438,Z 328.38,A -85,B 0,C 180,E1 23799.076,E2 23799.076} C_VEL
LIN {X 0,Y 640.838,Z 324.799,A -85,B 0,C 180,E1 23798.551,E2 23798.551} C_VEL
LIN {X 0,Y 640.831,Z 324.372,A -85,B 0,C 180,E1 23797.821,E2 23797.821} C_VEL
LIN {X 0,Y 640.779,Z 324.405,A -85,B 0,C 180,E1 23794.828,E2 23794.828} C_VEL
LIN {X 0,Y 640.83,Z 324.395,A -85,B 0,C 180,E1 23791.829,E2 23791.829} C_VEL
LIN {X 0,Y 640.788,Z 324.374,A -85,B 0,C 180,E1 23788.827,E2 23788.827} C_VEL
LIN {X 0,Y 640.829,Z 324.402,A -85,B 0,C 180,E1 23785.805,E2 23785.805} C_VEL
LIN {X 0,Y 640.796,Z 324.392,A -85,B 0,C 180,E1 23782.67,E2 23782.67} C_VEL
LIN {X 0,Y 640.825,Z 324.385,A -85,B 0,C 180,E1 23779.696,E2 23779.696} C_VEL
LIN {X 0,Y 640.807,Z 324.398,A -85,B 0,C 180,E1 23776.592,E2 23776.592} C_VEL
LIN {X 0,Y 640.819,Z 324.376,A -85,B 0,C 180,E1 23773.536,E2 23773.536} C_VEL
LIN {X 0,Y 640.812,Z 324.398,A -85,B 0,C 180,E1 23770.428,E2 23770.428} C_VEL
LIN {X 0,Y 640.812,Z 324.373,A -85,B 0,C 180,E1 23767.351,E2 23767.351} C_VEL
LIN {X 0,Y 640.817,Z 324.396,A -85,B 0,C 180,E1 23764.295,E2 23764.295} C_VEL
LIN {X 0,Y 640.805,Z 324.379,A -85,B 0,C 180,E1 23761.252,E2 23761.252} C_VEL
LIN {X 0,Y 640.824,Z 324.394,A -85,B 0,C 180,E1 23758.212,E2 23758.212} C_VEL
LIN {X 0,Y 640.8,Z 324.385,A -85,B 0,C 180,E1 23755.166,E2 23755.166} C_VEL
LIN {X 0,Y 640.829,Z 324.391,A -85,B 0,C 180,E1 23752.108,E2 23752.108} C_VEL
LIN {X 0,Y 640.792,Z 324.385,A -85,B 0,C 180,E1 23749.026,E2 23749.026} C_VEL
LIN {X 0,Y 640.831,Z 324.393,A -85,B 0,C 180,E1 23746.004,E2 23746.004} C_VEL
LIN {X 0,Y 640.783,Z 324.382,A -85,B 0,C 180,E1 23742.941,E2 23742.941} C_VEL
LIN {X 0,Y 640.827,Z 324.401,A -85,B 0,C 180,E1 23739.924,E2 23739.924} C_VEL
LIN {X 0,Y 640.774,Z 324.376,A -85,B 0,C 180,E1 23736.844,E2 23736.844} C_VEL
LIN {X 0,Y 640.813,Z 324.409,A -85,B 0,C 180,E1 23733.895,E2 23733.895} C_VEL
LIN {X 0,Y 640.77,Z 324.392,A -85,B 0,C 180,E1 23730.763,E2 23730.763} C_VEL
LIN {X 0,Y 640.773,Z 324.385,A -85,B 0,C 180,E1 23728.063,E2 23728.063} C_VEL
LIN {X 0,Y 640.776,Z 324.402,A -85,B 0,C 180,E1 23724.844,E2 23724.844} C_VEL
LIN {X 0,Y 640.826,Z 324.612,A -85,B 0,C 180,E1 23723.022,E2 23723.022} C_VEL
LIN {X 0,Y 642.291,Z 328.204,A -85,B 0,C 180,E1 23722.505,E2 23722.505} C_VEL
LIN {X 0,Y 643.605,Z 330.749,A -85,B 0,C 180,E1 23722.145,E2 23722.145} C_VEL
LIN {X 0,Y 645.979,Z 335.17,A -85,B 0,C 180,E1 23721.52,E2 23721.52} C_VEL
LIN {X 0,Y 653.846,Z 350.753,A -85,B 0,C 180,E1 23719.463,E2 23719.463} C_VEL
LIN {X 0,Y 656.072,Z 354.393,A -85,B 0,C 180,E1 23719.141,E2 23719.141} C_VEL
LIN {X 0,Y 671.533,Z 375.966,A -85,B 0,C 180,E1 23717.425,E2 23717.425} C_VEL
LIN {X 0,Y 672.775,Z 381.996,A -85,B 0,C 180,E1 23717.229,E2 23717.229} C_VEL
LIN {X 0,Y 669.057,Z 593.437,A -85,B 0,C 180,E1 23714.375,E2 23714.375} C_VEL
LIN {X 0,Y 665.411,Z 817.207,A -85,B 0,C 180,E1 23711.442,E2 23711.442} C_VEL
LIN {X 0,Y 664.554,Z 843.297,A -85,B 0,C 180,E1 23711.027,E2 23711.027} C_VEL
LIN {X 0,Y 663.545,Z 866.278,A -85,B 0,C 180,E1 23710.536,E2 23710.536} C_VEL
LIN {X 0,Y 662.199,Z 891.667,A -85,B 0,C 180,E1 23709.85,E2 23709.85} C_VEL
LIN {X 0,Y 660.422,Z 918.731,A -85,B 0,C 180,E1 23708.925,E2 23708.925} C_VEL
LIN {X 0,Y 658.813,Z 940.775,A -85,B 0,C 180,E1 23708.029,E2 23708.029} C_VEL
LIN {X 0,Y 657.176,Z 961.712,A -85,B 0,C 180,E1 23707.049,E2 23707.049} C_VEL
LIN {X 0,Y 655.151,Z 986.542,A -85,B 0,C 180,E1 23705.714,E2 23705.714} C_VEL
LIN {X 0,Y 653.094,Z 1009.33,A -85,B 0,C 180,E1 23704.291,E2 23704.291} C_VEL
LIN {X 0,Y 651.371,Z 1028.241,A -85,B 0,C 180,E1 23702.968,E2 23702.968} C_VEL
LIN {X 0,Y 649.557,Z 1048.292,A -85,B 0,C 180,E1 23701.403,E2 23701.403} C_VEL
LIN {X 0,Y 647.651,Z 1069.754,A -85,B 0,C 180,E1 23699.504,E2 23699.504} C_VEL
LIN {X 0,Y 646.219,Z 1086.384,A -85,B 0,C 180,E1 23697.857,E2 23697.857} C_VEL
LIN {X 0,Y 644.822,Z 1103.073,A -85,B 0,C 180,E1 23696.029,E2 23696.029} C_VEL
LIN {X 0,Y 643.432,Z 1121.565,A -85,B 0,C 180,E1 23693.733,E2 23693.733} C_VEL
LIN {X 0,Y 642.505,Z 1135.113,A -85,B 0,C 180,E1 23691.835,E2 23691.835} C_VEL
LIN {X 0,Y 641.693,Z 1148.368,A -85,B 0,C 180,E1 23689.752,E2 23689.752} C_VEL
LIN {X 0,Y 641.005,Z 1161.81,A -85,B 0,C 180,E1 23687.321,E2 23687.321} C_VEL
LIN {X 0,Y 640.57,Z 1171.57,A -85,B 0,C 180,E1 23685.277,E2 23685.277} C_VEL
LIN {X 0,Y 640.319,Z 1179.516,A -85,B 0,C 180,E1 23683.362,E2 23683.362} C_VEL
LIN {X 0,Y 640.102,Z 1187.237,A -85,B 0,C 180,E1 23681.189,E2 23681.189} C_VEL
LIN {X 0,Y 639.992,Z 1194.036,A -85,B 0,C 180,E1 23678.807,E2 23678.807} C_VEL
LIN {X 0,Y 639.936,Z 1199.169,A -85,B 0,C 180,E1 23676.412,E2 23676.412} C_VEL
LIN {X 0,Y 639.917,Z 1202.586,A -85,B 0,C 180,E1 23674.122,E2 23674.122} C_VEL
LIN {X 0,Y 639.908,Z 1204.578,A -85,B 0,C 180,E1 23671.701,E2 23671.701} C_VEL
LIN {X 0,Y 639.892,Z 1204.872,A -85,B 0,C 180,E1 23669.463,E2 23669.463} C_VEL
LIN {X 0,Y 639.91,Z 1203.941,A -85,B 0,C 180,E1 23667.313,E2 23667.313} C_VEL
LIN {X 0,Y 639.922,Z 1201.552,A -85,B 0,C 180,E1 23665.07,E2 23665.07} C_VEL
LIN {X 0,Y 639.954,Z 1197.346,A -85,B 0,C 180,E1 23662.639,E2 23662.639} C_VEL
LIN {X 0,Y 640.025,Z 1191.623,A -85,B 0,C 180,E1 23660.286,E2 23660.286} C_VEL
LIN {X 0,Y 640.164,Z 1184.589,A -85,B 0,C 180,E1 23658.01,E2 23658.01} C_VEL
LIN {X 0,Y 640.483,Z 1174.739,A -85,B 0,C 180,E1 23655.443,E2 23655.443} C_VEL
LIN {X 0,Y 640.844,Z 1164.999,A -85,B 0,C 180,E1 23653.316,E2 23653.316} C_VEL
LIN {X 0,Y 641.35,Z 1154.758,A -85,B 0,C 180,E1 23651.361,E2 23651.361} C_VEL
LIN {X 0,Y 642.054,Z 1142.527,A -85,B 0,C 180,E1 23649.298,E2 23649.298} C_VEL
LIN {X 0,Y 643.083,Z 1126.496,A -85,B 0,C 180,E1 23646.932,E2 23646.932} C_VEL
LIN {X 0,Y 644.145,Z 1111.852,A -85,B 0,C 180,E1 23645.025,E2 23645.025} C_VEL
LIN {X 0,Y 645.468,Z 1095.428,A -85,B 0,C 180,E1 23643.107,E2 23643.107} C_VEL
LIN {X 0,Y 647.157,Z 1075.328,A -85,B 0,C 180,E1 23641.029,E2 23641.029} C_VEL
LIN {X 0,Y 648.611,Z 1058.941,A -85,B 0,C 180,E1 23639.514,E2 23639.514} C_VEL
LIN {X 0,Y 650.172,Z 1041.615,A -85,B 0,C 180,E1 23638.06,E2 23638.06} C_VEL
LIN {X 0,Y 652.2,Z 1019.536,A -85,B 0,C 180,E1 23636.396,E2 23636.396} C_VEL
LIN {X 0,Y 654.206,Z 996.463,A -85,B 0,C 180,E1 23634.884,E2 23634.884} C_VEL
LIN {X 0,Y 655.998,Z 975.839,A -85,B 0,C 180,E1 23633.69,E2 23633.69} C_VEL
LIN {X 0,Y 657.989,Z 952.261,A -85,B 0,C 180,E1 23632.49,E2 23632.49} C_VEL
LIN {X 0,Y 659.919,Z 926.423,A -85,B 0,C 180,E1 23631.373,E2 23631.373} C_VEL
LIN {X 0,Y 661.331,Z 904.844,A -85,B 0,C 180,E1 23630.579,E2 23630.579} C_VEL
LIN {X 0,Y 662.659,Z 882.891,A -85,B 0,C 180,E1 23629.897,E2 23629.897} C_VEL
LIN {X 0,Y 663.968,Z 857.902,A -85,B 0,C 180,E1 23629.267,E2 23629.267} C_VEL
LIN {X 0,Y 665.055,Z 829.669,A -85,B 0,C 180,E1 23628.739,E2 23628.739} C_VEL
LIN {X 0,Y 666.571,Z 744.944,A -85,B 0,C 180,E1 23627.619,E2 23627.619} C_VEL
LIN {X 0,Y 670.285,Z 522.402,A -85,B 0,C 180,E1 23624.677,E2 23624.677} C_VEL
LIN {X 0,Y 672.653,Z 380.618,A -85,B 0,C 180,E1 23622.739,E2 23622.739} C_VEL
LIN {X 0,Y 671.298,Z 375.627,A -85,B 0,C 180,E1 23622.55,E2 23622.55} C_VEL
LIN {X 0,Y 656.073,Z 354.393,A -85,B 0,C 180,E1 23620.859,E2 23620.859} C_VEL
LIN {X 0,Y 654.197,Z 351.561,A -85,B 0,C 180,E1 23620.625,E2 23620.625} C_VEL
LIN {X 0,Y 648.637,Z 340.558,A -85,B 0,C 180,E1 23619.2,E2 23619.2} C_VEL
LIN {X 0,Y 644.823,Z 332.936,A -85,B 0,C 180,E1 23618.171,E2 23618.171} C_VEL
LIN {X 0,Y 642.288,Z 328.203,A -85,B 0,C 180,E1 23617.495,E2 23617.495} C_VEL
LIN {X 0,Y 640.824,Z 324.609,A -85,B 0,C 180,E1 23616.97,E2 23616.97} C_VEL
LIN {X 0,Y 640.762,Z 324.399,A -85,B 0,C 180,E1 23613.855,E2 23613.855} C_VEL
LIN {X 0,Y 640.783,Z 324.404,A -85,B 0,C 180,E1 23611.056,E2 23611.056} C_VEL
LIN {X 0,Y 640.775,Z 324.38,A -85,B 0,C 180,E1 23607.812,E2 23607.812} C_VEL
LIN {X 0,Y 640.79,Z 324.402,A -85,B 0,C 180,E1 23604.962,E2 23604.962} C_VEL
LIN {X 0,Y 640.787,Z 324.404,A -85,B 0,C 180,E1 23601.704,E2 23601.704} C_VEL
LIN {X 0,Y 640.796,Z 324.382,A -85,B 0,C 180,E1 23598.845,E2 23598.845} C_VEL
LIN {X 0,Y 640.802,Z 324.406,A -85,B 0,C 180,E1 23595.661,E2 23595.661} C_VEL
LIN {X 0,Y 640.803,Z 324.375,A -85,B 0,C 180,E1 23592.71,E2 23592.71} C_VEL
LIN {X 0,Y 640.807,Z 324.404,A -85,B 0,C 180,E1 23589.52,E2 23589.52} C_VEL
LIN {X 0,Y 640.822,Z 324.369,A -85,B 0,C 180,E1 23586.45,E2 23586.45} C_VEL
LIN {X 0,Y 640.805,Z 324.405,A -85,B 0,C 180,E1 23583.22,E2 23583.22} C_VEL
LIN {X 0,Y 640.823,Z 324.367,A -85,B 0,C 180,E1 23580.179,E2 23580.179} C_VEL
LIN {X 0,Y 640.808,Z 324.403,A -85,B 0,C 180,E1 23577.048,E2 23577.048} C_VEL
LIN {X 0,Y 640.816,Z 324.366,A -85,B 0,C 180,E1 23573.999,E2 23573.999} C_VEL
LIN {X 0,Y 640.814,Z 324.4,A -85,B 0,C 180,E1 23570.933,E2 23570.933} C_VEL
LIN {X 0,Y 640.809,Z 324.368,A -85,B 0,C 180,E1 23567.84,E2 23567.84} C_VEL
LIN {X 0,Y 640.82,Z 324.403,A -85,B 0,C 180,E1 23564.803,E2 23564.803} C_VEL
LIN {X 0,Y 640.803,Z 324.372,A -85,B 0,C 180,E1 23561.722,E2 23561.722} C_VEL
LIN {X 0,Y 640.825,Z 324.406,A -85,B 0,C 180,E1 23558.67,E2 23558.67} C_VEL
LIN {X 0,Y 640.797,Z 324.379,A -85,B 0,C 180,E1 23555.575,E2 23555.575} C_VEL
LIN {X 0,Y 640.827,Z 324.392,A -85,B 0,C 180,E1 23552.493,E2 23552.493} C_VEL
LIN {X 0,Y 640.792,Z 324.406,A -85,B 0,C 180,E1 23549.423,E2 23549.423} C_VEL
LIN {X 0,Y 640.827,Z 324.372,A -85,B 0,C 180,E1 23546.364,E2 23546.364} C_VEL
LIN {X 0,Y 640.782,Z 324.384,A -85,B 0,C 180,E1 23543.299,E2 23543.299} C_VEL
LIN {X 0,Y 640.823,Z 324.673,A -85,B 0,C 180,E1 23541.381,E2 23541.381} C_VEL
LIN {X 0,Y 642.134,Z 327.956,A -85,B 0,C 180,E1 23540.902,E2 23540.902} C_VEL
LIN {X 0,Y 643.465,Z 330.378,A -85,B 0,C 180,E1 23540.539,E2 23540.539} C_VEL
LIN {X 0,Y 648.002,Z 339.544,A -85,B 0,C 180,E1 23539.254,E2 23539.254} C_VEL
LIN {X 0,Y 654.355,Z 352.67,A -85,B 0,C 180,E1 23537.514,E2 23537.514} C_VEL
LIN {X 0,Y 654.855,Z 353.64,A -85,B 0,C 180,E1 23537.387,E2 23537.387} C_VEL
LIN {X 0,Y 656.453,Z 358.265,A -85,B 0,C 180,E1 23536.859,E2 23536.859} C_VEL
LIN {X 0,Y 656.921,Z 365.423,A -85,B 0,C 180,E1 23536.245,E2 23536.245} C_VEL
LIN {X 0,Y 655.849,Z 379.529,A -85,B 0,C 180,E1 23535.237,E2 23535.237} C_VEL
LIN {X 0,Y 654.888,Z 394.844,A -85,B 0,C 180,E1 23534.177,E2 23534.177} C_VEL
LIN {X 0,Y 661.76,Z 426.746,A -85,B 0,C 180,E1 23533.078,E2 23533.078} C_VEL
LIN {X 0,Y 657.406,Z 664.276,A -85,B 0,C 180,E1 23529.952,E2 23529.952} C_VEL
LIN {X 0,Y 654.258,Z 833.239,A -85,B 0,C 180,E1 23527.736,E2 23527.736} C_VEL
LIN {X 0,Y 653.26,Z 859.352,A -85,B 0,C 180,E1 23527.241,E2 23527.241} C_VEL
LIN {X 0,Y 652.23,Z 880.232,A -85,B 0,C 180,E1 23526.718,E2 23526.718} C_VEL
LIN {X 0,Y 651.109,Z 899.829,A -85,B 0,C 180,E1 23526.122,E2 23526.122} C_VEL
LIN {X 0,Y 649.741,Z 921.143,A -85,B 0,C 180,E1 23525.351,E2 23525.351} C_VEL
LIN {X 0,Y 647.927,Z 945.855,A -85,B 0,C 180,E1 23524.282,E2 23524.282} C_VEL
LIN {X 0,Y 646.303,Z 966.028,A -85,B 0,C 180,E1 23523.26,E2 23523.26} C_VEL
LIN {X 0,Y 644.543,Z 987.1,A -85,B 0,C 180,E1 23522.042,E2 23522.042} C_VEL
LIN {X 0,Y 642.596,Z 1009.646,A -85,B 0,C 180,E1 23520.533,E2 23520.533} C_VEL
LIN {X 0,Y 641.026,Z 1027.403,A -85,B 0,C 180,E1 23519.186,E2 23519.186} C_VEL
LIN {X 0,Y 639.36,Z 1046.407,A -85,B 0,C 180,E1 23517.575,E2 23517.575} C_VEL
LIN {X 0,Y 637.735,Z 1065.319,A -85,B 0,C 180,E1 23515.741,E2 23515.741} C_VEL
LIN {X 0,Y 636.519,Z 1080.365,A -85,B 0,C 180,E1 23514.106,E2 23514.106} C_VEL
LIN {X 0,Y 635.232,Z 1097.552,A -85,B 0,C 180,E1 23512.001,E2 23512.001} C_VEL
LIN {X 0,Y 634.277,Z 1111.126,A -85,B 0,C 180,E1 23510.1,E2 23510.1} C_VEL
LIN {X 0,Y 633.526,Z 1123.696,A -85,B 0,C 180,E1 23508.115,E2 23508.115} C_VEL
LIN {X 0,Y 632.873,Z 1136.467,A -85,B 0,C 180,E1 23505.768,E2 23505.768} C_VEL
LIN {X 0,Y 632.487,Z 1145.593,A -85,B 0,C 180,E1 23503.811,E2 23503.811} C_VEL
LIN {X 0,Y 632.212,Z 1154.461,A -85,B 0,C 180,E1 23501.587,E2 23501.587} C_VEL
LIN {X 0,Y 632.037,Z 1161.76,A -85,B 0,C 180,E1 23499.286,E2 23499.286} C_VEL
LIN {X 0,Y 631.961,Z 1166.64,A -85,B 0,C 180,E1 23497.363,E2 23497.363} C_VEL
LIN {X 0,Y 631.915,Z 1170.546,A -85,B 0,C 180,E1 23495.357,E2 23495.357} C_VEL
LIN {X 0,Y 631.906,Z 1173.563,A -85,B 0,C 180,E1 23492.993,E2 23492.993} C_VEL
LIN {X 0,Y 631.905,Z 1174.769,A -85,B 0,C 180,E1 23490.907,E2 23490.907} C_VEL
LIN {X 0,Y 631.909,Z 1174.77,A -85,B 0,C 180,E1 23489.003,E2 23489.003} C_VEL
LIN {X 0,Y 631.908,Z 1173.566,A -85,B 0,C 180,E1 23486.916,E2 23486.916} C_VEL
LIN {X 0,Y 631.916,Z 1170.543,A -85,B 0,C 180,E1 23484.552,E2 23484.552} C_VEL
LIN {X 0,Y 631.955,Z 1166.637,A -85,B 0,C 180,E1 23482.546,E2 23482.546} C_VEL
LIN {X 0,Y 632.04,Z 1161.756,A -85,B 0,C 180,E1 23480.622,E2 23480.622} C_VEL
LIN {X 0,Y 632.212,Z 1154.454,A -85,B 0,C 180,E1 23478.321,E2 23478.321} C_VEL
LIN {X 0,Y 632.487,Z 1145.547,A -85,B 0,C 180,E1 23476.089,E2 23476.089} C_VEL
LIN {X 0,Y 632.859,Z 1136.734,A -85,B 0,C 180,E1 23474.196,E2 23474.196} C_VEL
LIN {X 0,Y 633.466,Z 1124.817,A -85,B 0,C 180,E1 23471.979,E2 23471.979} C_VEL
LIN {X 0,Y 634.232,Z 1111.725,A -85,B 0,C 180,E1 23469.899,E2 23469.899} C_VEL
LIN {X 0,Y 635.181,Z 1098.211,A -85,B 0,C 180,E1 23467.998,E2 23467.998} C_VEL
LIN {X 0,Y 636.452,Z 1081.141,A -85,B 0,C 180,E1 23465.892,E2 23465.892} C_VEL
LIN {X 0,Y 637.706,Z 1065.693,A -85,B 0,C 180,E1 23464.209,E2 23464.209} C_VEL
LIN {X 0,Y 639.329,Z 1046.856,A -85,B 0,C 180,E1 23462.373,E2 23462.373} C_VEL
LIN {X 0,Y 641.028,Z 1027.366,A -85,B 0,C 180,E1 23460.72,E2 23460.72} C_VEL
LIN {X 0,Y 642.67,Z 1008.81,A -85,B 0,C 180,E1 23459.316,E2 23459.316} C_VEL
LIN {X 0,Y 644.693,Z 985.263,A -85,B 0,C 180,E1 23457.757,E2 23457.757} C_VEL
LIN {X 0,Y 646.406,Z 964.861,A -85,B 0,C 180,E1 23456.587,E2 23456.587} C_VEL
LIN {X 0,Y 648.304,Z 941.496,A -85,B 0,C 180,E1 23455.42,E2 23455.42} C_VEL
LIN {X 0,Y 649.925,Z 918.1,A -85,B 0,C 180,E1 23454.442,E2 23454.442} C_VEL
LIN {X 0,Y 651.238,Z 897.585,A -85,B 0,C 180,E1 23453.714,E2 23453.714} C_VEL
LIN {X 0,Y 652.504,Z 875.179,A -85,B 0,C 180,E1 23453.05,E2 23453.05} C_VEL
LIN {X 0,Y 653.667,Z 848.556,A -85,B 0,C 180,E1 23452.442,E2 23452.442} C_VEL
LIN {X 0,Y 654.442,Z 825.464,A -85,B 0,C 180,E1 23452.059,E2 23452.059} C_VEL
LIN {X 0,Y 658.775,Z 590.472,A -85,B 0,C 180,E1 23448.991,E2 23448.991} C_VEL
LIN {X 0,Y 661.671,Z 426.096,A -85,B 0,C 180,E1 23446.814,E2 23446.814} C_VEL
LIN {X 0,Y 654.818,Z 394.201,A -85,B 0,C 180,E1 23445.704,E2 23445.704} C_VEL
LIN {X 0,Y 656.165,Z 374.656,A -85,B 0,C 180,E1 23444.322,E2 23444.322} C_VEL
LIN {X 0,Y 647.556,Z 355.631,A -85,B 0,C 180,E1 23441.959,E2 23441.959} C_VEL
LIN {X 0,Y 640.928,Z 342.101,A -85,B 0,C 180,E1 23440.114,E2 23440.114} C_VEL
LIN {X 0,Y 636.748,Z 333.792,A -85,B 0,C 180,E1 23438.912,E2 23438.912} C_VEL
LIN {X 0,Y 634.565,Z 329.414,A -85,B 0,C 180,E1 23438.262,E2 23438.262} C_VEL
LIN {X 0,Y 632.921,Z 325.594,A -85,B 0,C 180,E1 23437.665,E2 23437.665} C_VEL
LIN {X 0,Y 632.84,Z 325.386,A -85,B 0,C 180,E1 23434.667,E2 23434.667} C_VEL
LIN {X 0,Y 632.893,Z 325.389,A -85,B 0,C 180,E1 23431.621,E2 23431.621} C_VEL
LIN {X 0,Y 632.845,Z 325.362,A -85,B 0,C 180,E1 23428.603,E2 23428.603} C_VEL
LIN {X 0,Y 632.889,Z 325.385,A -85,B 0,C 180,E1 23425.551,E2 23425.551} C_VEL
LIN {X 0,Y 632.856,Z 325.382,A -85,B 0,C 180,E1 23422.442,E2 23422.442} C_VEL
LIN {X 0,Y 632.882,Z 325.367,A -85,B 0,C 180,E1 23419.377,E2 23419.377} C_VEL
LIN {X 0,Y 632.866,Z 325.391,A -85,B 0,C 180,E1 23416.239,E2 23416.239} C_VEL
LIN {X 0,Y 632.878,Z 325.357,A -85,B 0,C 180,E1 23413.15,E2 23413.15} C_VEL
LIN {X 0,Y 632.876,Z 325.391,A -85,B 0,C 180,E1 23410.008,E2 23410.008} C_VEL
LIN {X 0,Y 632.883,Z 325.351,A -85,B 0,C 180,E1 23406.805,E2 23406.805} C_VEL
LIN {X 0,Y 632.883,Z 325.398,A -85,B 0,C 180,E1 23403.533,E2 23403.533} C_VEL
LIN {X 0,Y 632.884,Z 325.352,A -85,B 0,C 180,E1 23400.362,E2 23400.362} C_VEL
LIN {X 0,Y 632.866,Z 325.399,A -85,B 0,C 180,E1 23397.193,E2 23397.193} C_VEL
LIN {X 0,Y 632.883,Z 325.355,A -85,B 0,C 180,E1 23394.106,E2 23394.106} C_VEL
LIN {X 0,Y 632.856,Z 325.397,A -85,B 0,C 180,E1 23391.001,E2 23391.001} C_VEL
LIN {X 0,Y 632.887,Z 325.354,A -85,B 0,C 180,E1 23387.941,E2 23387.941} C_VEL
LIN {X 0,Y 632.848,Z 325.399,A -85,B 0,C 180,E1 23384.874,E2 23384.874} C_VEL
LIN {X 0,Y 632.888,Z 325.355,A -85,B 0,C 180,E1 23381.866,E2 23381.866} C_VEL
LIN {X 0,Y 632.841,Z 325.396,A -85,B 0,C 180,E1 23378.778,E2 23378.778} C_VEL
LIN {X 0,Y 632.89,Z 325.367,A -85,B 0,C 180,E1 23375.724,E2 23375.724} C_VEL
LIN {X 0,Y 632.831,Z 325.376,A -85,B 0,C 180,E1 23372.728,E2 23372.728} C_VEL
LIN {X 0,Y 632.866,Z 325.397,A -85,B 0,C 180,E1 23369.84,E2 23369.84} C_VEL
LIN {X 0,Y 632.824,Z 325.372,A -85,B 0,C 180,E1 23366.702,E2 23366.702} C_VEL
LIN {X 0,Y 632.859,Z 325.557,A -85,B 0,C 180,E1 23363.891,E2 23363.891} C_VEL
LIN {X 0,Y 634.324,Z 329.033,A -85,B 0,C 180,E1 23363.353,E2 23363.353} C_VEL
LIN {X 0,Y 635.441,Z 331,A -85,B 0,C 180,E1 23363.052,E2 23363.052} C_VEL
LIN {X 0,Y 642.056,Z 343.75,A -85,B 0,C 180,E1 23361.241,E2 23361.241} C_VEL
LIN {X 0,Y 646.613,Z 352.704,A -85,B 0,C 180,E1 23360.078,E2 23360.078} C_VEL
LIN {X 0,Y 664.099,Z 377.482,A -85,B 0,C 180,E1 23358.048,E2 23358.048} C_VEL
LIN {X 0,Y 666.593,Z 381.217,A -85,B 0,C 180,E1 23357.771,E2 23357.771} C_VEL
LIN {X 0,Y 667.049,Z 384.306,A -85,B 0,C 180,E1 23357.684,E2 23357.684} C_VEL
LIN {X 0,Y 664.115,Z 551.629,A -85,B 0,C 180,E1 23355.421,E2 23355.421} C_VEL
LIN {X 0,Y 660.079,Z 778.443,A -85,B 0,C 180,E1 23352.412,E2 23352.412} C_VEL
LIN {X 0,Y 658.968,Z 832.18,A -85,B 0,C 180,E1 23351.684,E2 23351.684} C_VEL
LIN {X 0,Y 657.733,Z 860.263,A -85,B 0,C 180,E1 23351.137,E2 23351.137} C_VEL
LIN {X 0,Y 656.432,Z 883.654,A -85,B 0,C 180,E1 23350.536,E2 23350.536} C_VEL
LIN {X 0,Y 654.997,Z 905.876,A -85,B 0,C 180,E1 23349.838,E2 23349.838} C_VEL
LIN {X 0,Y 653.196,Z 931.52,A -85,B 0,C 180,E1 23348.873,E2 23348.873} C_VEL
LIN {X 0,Y 651.036,Z 956.893,A -85,B 0,C 180,E1 23347.724,E2 23347.724} C_VEL
LIN {X 0,Y 649.169,Z 977.833,A -85,B 0,C 180,E1 23346.632,E2 23346.632} C_VEL
LIN {X 0,Y 647.121,Z 999.851,A -85,B 0,C 180,E1 23345.33,E2 23345.33} C_VEL
LIN {X 0,Y 644.785,Z 1024.233,A -85,B 0,C 180,E1 23343.668,E2 23343.668} C_VEL
LIN {X 0,Y 642.958,Z 1042.837,A -85,B 0,C 180,E1 23342.236,E2 23342.236} C_VEL
LIN {X 0,Y 641.226,Z 1060.716,A -85,B 0,C 180,E1 23340.709,E2 23340.709} C_VEL
LIN {X 0,Y 639.242,Z 1081.496,A -85,B 0,C 180,E1 23338.724,E2 23338.724} C_VEL
LIN {X 0,Y 637.684,Z 1098.845,A -85,B 0,C 180,E1 23336.845,E2 23336.845} C_VEL
LIN {X 0,Y 636.316,Z 1114.6,A -85,B 0,C 180,E1 23334.949,E2 23334.949} C_VEL
LIN {X 0,Y 634.989,Z 1131.893,A -85,B 0,C 180,E1 23332.595,E2 23332.595} C_VEL
LIN {X 0,Y 634.107,Z 1144.858,A -85,B 0,C 180,E1 23330.587,E2 23330.587} C_VEL
LIN {X 0,Y 633.408,Z 1156.308,A -85,B 0,C 180,E1 23328.594,E2 23328.594} C_VEL
LIN {X 0,Y 632.814,Z 1168.201,A -85,B 0,C 180,E1 23326.24,E2 23326.24} C_VEL
LIN {X 0,Y 632.401,Z 1178.185,A -85,B 0,C 180,E1 23323.88,E2 23323.88} C_VEL
LIN {X 0,Y 632.166,Z 1185.9,A -85,B 0,C 180,E1 23321.743,E2 23321.743} C_VEL
LIN {X 0,Y 632.021,Z 1192.865,A -85,B 0,C 180,E1 23319.378,E2 23319.378} C_VEL
LIN {X 0,Y 631.94,Z 1198.423,A -85,B 0,C 180,E1 23316.906,E2 23316.906} C_VEL
LIN {X 0,Y 631.913,Z 1202.016,A -85,B 0,C 180,E1 23314.628,E2 23314.628} C_VEL
LIN {X 0,Y 631.91,Z 1204.211,A -85,B 0,C 180,E1 23312.358,E2 23312.358} C_VEL
LIN {X 0,Y 631.902,Z 1204.961,A -85,B 0,C 180,E1 23309.818,E2 23309.818} C_VEL
LIN {X 0,Y 631.908,Z 1204.075,A -85,B 0,C 180,E1 23307.46,E2 23307.46} C_VEL
LIN {X 0,Y 631.917,Z 1201.788,A -85,B 0,C 180,E1 23305.189,E2 23305.189} C_VEL
LIN {X 0,Y 631.957,Z 1197.734,A -85,B 0,C 180,E1 23302.728,E2 23302.728} C_VEL
LIN {X 0,Y 632.033,Z 1191.874,A -85,B 0,C 180,E1 23300.254,E2 23300.254} C_VEL
LIN {X 0,Y 632.182,Z 1184.889,A -85,B 0,C 180,E1 23297.949,E2 23297.949} C_VEL
LIN {X 0,Y 632.528,Z 1175.143,A -85,B 0,C 180,E1 23295.349,E2 23295.349} C_VEL
LIN {X 0,Y 632.943,Z 1164.997,A -85,B 0,C 180,E1 23293.102,E2 23293.102} C_VEL
LIN {X 0,Y 633.495,Z 1154.76,A -85,B 0,C 180,E1 23291.121,E2 23291.121} C_VEL
LIN {X 0,Y 634.298,Z 1141.946,A -85,B 0,C 180,E1 23288.936,E2 23288.936} C_VEL
LIN {X 0,Y 635.436,Z 1125.793,A -85,B 0,C 180,E1 23286.54,E2 23286.54} C_VEL
LIN {X 0,Y 636.63,Z 1111.077,A -85,B 0,C 180,E1 23284.61,E2 23284.61} C_VEL
LIN {X 0,Y 638.206,Z 1092.836,A -85,B 0,C 180,E1 23282.47,E2 23282.47} C_VEL
LIN {X 0,Y 639.97,Z 1073.807,A -85,B 0,C 180,E1 23280.518,E2 23280.518} C_VEL
LIN {X 0,Y 641.533,Z 1057.513,A -85,B 0,C 180,E1 23279.007,E2 23279.007} C_VEL
LIN {X 0,Y 643.322,Z 1039.179,A -85,B 0,C 180,E1 23277.468,E2 23277.468} C_VEL
LIN {X 0,Y 645.644,Z 1015.178,A -85,B 0,C 180,E1 23275.687,E2 23275.687} C_VEL
LIN {X 0,Y 647.618,Z 994.618,A -85,B 0,C 180,E1 23274.35,E2 23274.35} C_VEL
LIN {X 0,Y 649.502,Z 974.418,A -85,B 0,C 180,E1 23273.181,E2 23273.181} C_VEL
LIN {X 0,Y 651.752,Z 949.299,A -85,B 0,C 180,E1 23271.909,E2 23271.909} C_VEL
LIN {X 0,Y 653.675,Z 924.58,A -85,B 0,C 180,E1 23270.853,E2 23270.853} C_VEL
LIN {X 0,Y 655.117,Z 904.102,A -85,B 0,C 180,E1 23270.103,E2 23270.103} C_VEL
LIN {X 0,Y 656.515,Z 882.346,A -85,B 0,C 180,E1 23269.427,E2 23269.427} C_VEL
LIN {X 0,Y 657.912,Z 857.306,A -85,B 0,C 180,E1 23268.795,E2 23268.795} C_VEL
LIN {X 0,Y 659.041,Z 829.318,A -85,B 0,C 180,E1 23268.273,E2 23268.273} C_VEL
LIN {X 0,Y 660.709,Z 741.978,A -85,B 0,C 180,E1 23267.11,E2 23267.11} C_VEL
LIN {X 0,Y 664.699,Z 520.239,A -85,B 0,C 180,E1 23264.155,E2 23264.155} C_VEL
LIN {X 0,Y 666.97,Z 382.838,A -85,B 0,C 180,E1 23262.287,E2 23262.287} C_VEL
LIN {X 0,Y 666.119,Z 380.19,A -85,B 0,C 180,E1 23262.172,E2 23262.172} C_VEL
LIN {X 0,Y 648.349,Z 355.327,A -85,B 0,C 180,E1 23260.139,E2 23260.139} C_VEL
LIN {X 0,Y 646.152,Z 351.881,A -85,B 0,C 180,E1 23259.84,E2 23259.84} C_VEL
LIN {X 0,Y 639.358,Z 338.596,A -85,B 0,C 180,E1 23258.038,E2 23258.038} C_VEL
LIN {X 0,Y 635.369,Z 330.796,A -85,B 0,C 180,E1 23256.923,E2 23256.923} C_VEL
LIN {X 0,Y 632.921,Z 325.878,A -85,B 0,C 180,E1 23256.186,E2 23256.186} C_VEL
LIN {X 0,Y 632.812,Z 325.376,A -85,B 0,C 180,E1 23255.665,E2 23255.665} C_VEL
LIN {X 0,Y 632.871,Z 325.361,A -85,B 0,C 180,E1 23252.806,E2 23252.806} C_VEL
LIN {X 0,Y 632.829,Z 325.394,A -85,B 0,C 180,E1 23249.744,E2 23249.744} C_VEL
LIN {X 0,Y 632.85,Z 325.38,A -85,B 0,C 180,E1 23246.966,E2 23246.966} C_VEL
LIN {X 0,Y 632.842,Z 325.364,A -85,B 0,C 180,E1 23243.76,E2 23243.76} C_VEL
LIN {X 0,Y 632.865,Z 325.398,A -85,B 0,C 180,E1 23240.823,E2 23240.823} C_VEL
LIN {X 0,Y 632.853,Z 325.36,A -85,B 0,C 180,E1 23237.659,E2 23237.659} C_VEL
LIN {X 0,Y 632.876,Z 325.397,A -85,B 0,C 180,E1 23234.643,E2 23234.643} C_VEL
LIN {X 0,Y 632.857,Z 325.363,A -85,B 0,C 180,E1 23231.483,E2 23231.483} C_VEL
LIN {X 0,Y 632.887,Z 325.39,A -85,B 0,C 180,E1 23228.449,E2 23228.449} C_VEL
LIN {X 0,Y 632.859,Z 325.365,A -85,B 0,C 180,E1 23225.258,E2 23225.258} C_VEL
LIN {X 0,Y 632.887,Z 325.389,A -85,B 0,C 180,E1 23222.173,E2 23222.173} C_VEL
LIN {X 0,Y 632.864,Z 325.36,A -85,B 0,C 180,E1 23219.095,E2 23219.095} C_VEL
LIN {X 0,Y 632.881,Z 325.389,A -85,B 0,C 180,E1 23216.014,E2 23216.014} C_VEL
LIN {X 0,Y 632.869,Z 325.355,A -85,B 0,C 180,E1 23212.921,E2 23212.921} C_VEL
LIN {X 0,Y 632.875,Z 325.389,A -85,B 0,C 180,E1 23209.827,E2 23209.827} C_VEL
LIN {X 0,Y 632.873,Z 325.358,A -85,B 0,C 180,E1 23206.711,E2 23206.711} C_VEL
LIN {X 0,Y 632.869,Z 325.39,A -85,B 0,C 180,E1 23203.666,E2 23203.666} C_VEL
LIN {X 0,Y 632.879,Z 325.368,A -85,B 0,C 180,E1 23200.527,E2 23200.527} C_VEL
LIN {X 0,Y 632.859,Z 325.383,A -85,B 0,C 180,E1 23197.521,E2 23197.521} C_VEL
LIN {X 0,Y 632.886,Z 325.385,A -85,B 0,C 180,E1 23194.437,E2 23194.437} C_VEL
LIN {X 0,Y 632.851,Z 325.361,A -85,B 0,C 180,E1 23191.397,E2 23191.397} C_VEL
LIN {X 0,Y 632.892,Z 325.391,A -85,B 0,C 180,E1 23188.364,E2 23188.364} C_VEL
LIN {X 0,Y 632.847,Z 325.385,A -85,B 0,C 180,E1 23185.244,E2 23185.244} C_VEL
LIN {X 0,Y 632.92,Z 325.575,A -85,B 0,C 180,E1 23182.239,E2 23182.239} C_VEL
LIN {X 0,Y 634.267,Z 328.986,A -85,B 0,C 180,E1 23181.717,E2 23181.717} C_VEL
LIN {X 0,Y 635.53,Z 331.433,A -85,B 0,C 180,E1 23181.346,E2 23181.346} C_VEL
LIN {X 0,Y 639.859,Z 339.821,A -85,B 0,C 180,E1 23180.109,E2 23180.109} C_VEL
LIN {X 0,Y 646.646,Z 353.912,A -85,B 0,C 180,E1 23178.185,E2 23178.185} C_VEL
LIN {X 0,Y 653.892,Z 369.588,A -85,B 0,C 180,E1 23176.199,E2 23176.199} C_VEL
LIN {X 0,Y 656.171,Z 375.05,A -85,B 0,C 180,E1 23175.557,E2 23175.557} C_VEL
LIN {X 0,Y 655.849,Z 379.529,A -85,B 0,C 180,E1 23175.237,E2 23175.237} C_VEL
LIN {X 0,Y 654.78,Z 383.947,A -85,B 0,C 180,E1 23174.998,E2 23174.998} C_VEL
LIN {X 0,Y 651,Z 393.538,A -85,B 0,C 180,E1 23174.723,E2 23174.723} C_VEL
LIN {X 0,Y 650.05,Z 399.247,A -85,B 0,C 180,E1 23174.573,E2 23174.573} C_VEL
LIN {X 0,Y 650.304,Z 401.327,A -85,B 0,C 180,E1 23174.502,E2 23174.502} C_VEL
LIN {X 0,Y 656.095,Z 428.855,A -85,B 0,C 180,E1 23173.549,E2 23173.549} C_VEL
LIN {X 0,Y 651.543,Z 665.86,A -85,B 0,C 180,E1 23170.415,E2 23170.415} C_VEL
LIN {X 0,Y 648.237,Z 830.043,A -85,B 0,C 180,E1 23168.246,E2 23168.246} C_VEL
LIN {X 0,Y 647.173,Z 856.191,A -85,B 0,C 180,E1 23167.763,E2 23167.763} C_VEL
LIN {X 0,Y 645.78,Z 881.277,A -85,B 0,C 180,E1 23167.126,E2 23167.126} C_VEL
LIN {X 0,Y 644.117,Z 907.518,A -85,B 0,C 180,E1 23166.289,E2 23166.289} C_VEL
LIN {X 0,Y 642.282,Z 931.621,A -85,B 0,C 180,E1 23165.338,E2 23165.338} C_VEL
LIN {X 0,Y 640.658,Z 951.892,A -85,B 0,C 180,E1 23164.401,E2 23164.401} C_VEL
LIN {X 0,Y 638.715,Z 974.94,A -85,B 0,C 180,E1 23163.17,E2 23163.17} C_VEL
LIN {X 0,Y 636.733,Z 996.302,A -85,B 0,C 180,E1 23161.836,E2 23161.836} C_VEL
LIN {X 0,Y 635.038,Z 1014.327,A -85,B 0,C 180,E1 23160.569,E2 23160.569} C_VEL
LIN {X 0,Y 633.044,Z 1035.329,A -85,B 0,C 180,E1 23158.903,E2 23158.903} C_VEL
LIN {X 0,Y 631.314,Z 1053.606,A -85,B 0,C 180,E1 23157.24,E2 23157.24} C_VEL
LIN {X 0,Y 629.846,Z 1069.951,A -85,B 0,C 180,E1 23155.582,E2 23155.582} C_VEL
LIN {X 0,Y 628.251,Z 1088.477,A -85,B 0,C 180,E1 23153.446,E2 23153.446} C_VEL
LIN {X 0,Y 627.128,Z 1102.481,A -85,B 0,C 180,E1 23151.611,E2 23151.611} C_VEL
LIN {X 0,Y 626.086,Z 1117.363,A -85,B 0,C 180,E1 23149.401,E2 23149.401} C_VEL
LIN {X 0,Y 625.337,Z 1129.561,A -85,B 0,C 180,E1 23147.302,E2 23147.302} C_VEL
LIN {X 0,Y 624.789,Z 1140.229,A -85,B 0,C 180,E1 23145.198,E2 23145.198} C_VEL
LIN {X 0,Y 624.362,Z 1150.593,A -85,B 0,C 180,E1 23142.763,E2 23142.763} C_VEL
LIN {X 0,Y 624.136,Z 1157.537,A -85,B 0,C 180,E1 23140.803,E2 23140.803} C_VEL
LIN {X 0,Y 624.009,Z 1163.798,A -85,B 0,C 180,E1 23138.663,E2 23138.663} C_VEL
LIN {X 0,Y 623.943,Z 1169.109,A -85,B 0,C 180,E1 23136.256,E2 23136.256} C_VEL
LIN {X 0,Y 623.912,Z 1172.234,A -85,B 0,C 180,E1 23134.228,E2 23134.228} C_VEL
LIN {X 0,Y 623.914,Z 1174.107,A -85,B 0,C 180,E1 23132.296,E2 23132.296} C_VEL
LIN {X 0,Y 623.916,Z 1174.993,A -85,B 0,C 180,E1 23130,E2 23130} C_VEL
LIN {X 0,Y 623.913,Z 1174.175,A -85,B 0,C 180,E1 23127.704,E2 23127.704} C_VEL
LIN {X 0,Y 623.911,Z 1172.347,A -85,B 0,C 180,E1 23125.773,E2 23125.773} C_VEL
LIN {X 0,Y 623.941,Z 1169.266,A -85,B 0,C 180,E1 23123.744,E2 23123.744} C_VEL
LIN {X 0,Y 624,Z 1164.044,A -85,B 0,C 180,E1 23121.337,E2 23121.337} C_VEL
LIN {X 0,Y 624.13,Z 1157.829,A -85,B 0,C 180,E1 23119.197,E2 23119.197} C_VEL
LIN {X 0,Y 624.35,Z 1150.915,A -85,B 0,C 180,E1 23117.232,E2 23117.232} C_VEL
LIN {X 0,Y 624.744,Z 1141.494,A -85,B 0,C 180,E1 23114.973,E2 23114.973} C_VEL
LIN {X 0,Y 625.306,Z 1130.046,A -85,B 0,C 180,E1 23112.698,E2 23112.698} C_VEL
LIN {X 0,Y 626.004,Z 1118.486,A -85,B 0,C 180,E1 23110.693,E2 23110.693} C_VEL
LIN {X 0,Y 627.077,Z 1103.126,A -85,B 0,C 180,E1 23108.388,E2 23108.388} C_VEL
LIN {X 0,Y 628.194,Z 1089.175,A -85,B 0,C 180,E1 23106.552,E2 23106.552} C_VEL
LIN {X 0,Y 629.621,Z 1072.637,A -85,B 0,C 180,E1 23104.61,E2 23104.61} C_VEL
LIN {X 0,Y 631.236,Z 1054.51,A -85,B 0,C 180,E1 23102.757,E2 23102.757} C_VEL
LIN {X 0,Y 632.84,Z 1037.407,A -85,B 0,C 180,E1 23101.191,E2 23101.191} C_VEL
LIN {X 0,Y 634.935,Z 1015.489,A -85,B 0,C 180,E1 23099.426,E2 23099.426} C_VEL
LIN {X 0,Y 636.697,Z 996.695,A -85,B 0,C 180,E1 23098.1,E2 23098.1} C_VEL
LIN {X 0,Y 638.583,Z 976.305,A -85,B 0,C 180,E1 23096.823,E2 23096.823} C_VEL
LIN {X 0,Y 640.606,Z 952.573,A -85,B 0,C 180,E1 23095.542,E2 23095.542} C_VEL
LIN {X 0,Y 642.216,Z 932.453,A -85,B 0,C 180,E1 23094.608,E2 23094.608} C_VEL
LIN {X 0,Y 643.949,Z 909.543,A -85,B 0,C 180,E1 23093.695,E2 23093.695} C_VEL
LIN {X 0,Y 645.679,Z 882.842,A -85,B 0,C 180,E1 23092.83,E2 23092.83} C_VEL
LIN {X 0,Y 646.915,Z 860.854,A -85,B 0,C 180,E1 23092.258,E2 23092.258} C_VEL
LIN {X 0,Y 648.1,Z 835.934,A -85,B 0,C 180,E1 23091.754,E2 23091.754} C_VEL
LIN {X 0,Y 649.165,Z 789.607,A -85,B 0,C 180,E1 23091.116,E2 23091.116} C_VEL
LIN {X 0,Y 653.448,Z 567.325,A -85,B 0,C 180,E1 23088.193,E2 23088.193} C_VEL
LIN {X 0,Y 655.998,Z 427.971,A -85,B 0,C 180,E1 23086.338,E2 23086.338} C_VEL
LIN {X 0,Y 648.718,Z 393.673,A -85,B 0,C 180,E1 23085.121,E2 23085.121} C_VEL
LIN {X 0,Y 649.829,Z 378.848,A -85,B 0,C 180,E1 23084.064,E2 23084.064} C_VEL
